KUKA KRL program: MyProgram_308().src

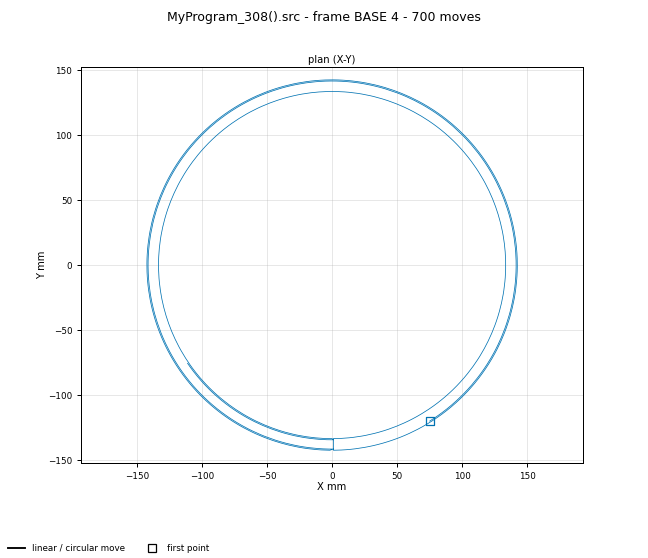
[picture p0: tool path of MyProgram_308().src in frame BASE 4, 700 of 700 moves have a stored position in this frame; points joined in program order, loops and branches not executed]
&ACCESS RVP
&REL 1
&PARAM TEMPLATE = C:\KRC\Roboter\Template\vorgabe
&PARAM EDITMASK = *
DEF MyProgram_308()
; ---- Setting reference (Base) ----
$BASE = BASE_DATA[4]

; --------------------------
; ---- Setting tool (TCP) ----
$TOOL = TOOL_DATA[3]
; --------------------------

$VEL.CP = VEL_APROX_PRINT
Startdeposition()
$VEL.CP = VEL_PRINT
LIN {X 75.0698,Y -120.0546,Z 181,A -53.2444,B 4.6912,C 0.3512,E1 4.792,E2 505.9034} C_DIS
LIN {X 78.7093,Y -117.7003,Z 181,A -51.6631,B 4.6912,C 0.3506,E1 4.7956,E2 504.3443} C_DIS
LIN {X 81.6771,Y -115.6604,Z 181,A -50.1341,B 4.6915,C 0.3471,E1 4.7991,E2 502.8043} C_DIS
LIN {X 84.8827,Y -113.3295,Z 181,A -48.4927,B 4.6918,C 0.3438,E1 4.8028,E2 501.1565} C_DIS
LIN {X 88.5091,Y -110.5206,Z 181,A -46.7634,B 4.6918,C 0.342,E1 4.8066,E2 499.443} C_DIS
LIN {X 91.7786,Y -107.8201,Z 181,A -44.9889,B 4.6922,C 0.338,E1 4.8104,E2 497.659} C_DIS
LIN {X 95.3898,Y -104.6393,Z 181,A -43.0975,B 4.6924,C 0.3349,E1 4.8143,E2 495.7737} C_DIS
LIN {X 98.6334,Y -101.5873,Z 181,A -41.3388,B 4.6926,C 0.3318,E1 4.8179,E2 494.0193} C_DIS
LIN {X 101.7844,Y -98.4298,Z 181,A -39.801,B 4.6926,C 0.3316,E1 4.8208,E2 492.5162} C_DIS
LIN {X 104.4298,Y -95.6189,Z 181,A -38.0744,B 4.693,C 0.326,E1 4.8242,E2 490.766} C_DIS
LIN {X 107.3448,Y -92.334,Z 181,A -36.3549,B 4.6932,C 0.3229,E1 4.8273,E2 489.0528} C_DIS
LIN {X 110.0788,Y -89.0572,Z 181,A -34.8071,B 4.6933,C 0.3214,E1 4.83,E2 487.5278} C_DIS
LIN {X 111.9572,Y -86.6838,Z 181,A -33.148,B 4.6939,C 0.3127,E1 4.833,E2 485.8087} C_DIS
LIN {X 114.3083,Y -83.5596,Z 181,A -31.9004,B 4.6939,C 0.3136,E1 4.8349,E2 484.6052} C_DIS
LIN {X 116.9623,Y -79.8026,Z 181,A -30.0572,B 4.6942,C 0.3094,E1 4.8379,E2 482.7628} C_DIS
LIN {X 119.4438,Y -76.0381,Z 181,A -28.3668,B 4.6943,C 0.3068,E1 4.8404,E2 481.0891} C_DIS
LIN {X 122.1556,Y -71.5997,Z 181,A -26.2713,B 4.6946,C 0.3017,E1 4.8434,E2 478.993} C_DIS
LIN {X 124.3843,Y -67.654,Z 181,A -24.4934,B 4.6949,C 0.2979,E1 4.8458,E2 477.2211} C_DIS
LIN {X 125.8992,Y -64.7895,Z 181,A -23.2049,B 4.6951,C 0.2948,E1 4.8475,E2 475.9344} C_DIS
LIN {X 127.5298,Y -61.5171,Z 181,A -21.7796,B 4.6953,C 0.2917,E1 4.8492,E2 474.5151} C_DIS
LIN {X 129.1189,Y -58.1061,Z 181,A -20.448,B 4.6953,C 0.2904,E1 4.8508,E2 473.2081} C_DIS
LIN {X 130.2583,Y -55.509,Z 181,A -19.102,B 4.6957,C 0.2846,E1 4.8523,E2 471.8344} C_DIS
LIN {X 131.8713,Y -51.5555,Z 181,A -17.5331,B 4.6959,C 0.2823,E1 4.8539,E2 470.2854} C_DIS
LIN {X 132.9031,Y -48.8412,Z 181,A -16.3204,B 4.6961,C 0.2786,E1 4.8551,E2 469.0666} C_DIS
LIN {X 134.269,Y -44.9427,Z 181,A -14.7391,B 4.6963,C 0.2753,E1 4.8565,E2 467.496} C_DIS
LIN {X 136.3041,Y -38.3301,Z 181,A -12.0529,B 4.6966,C 0.2692,E1 4.8586,E2 464.8228} C_DIS
LIN {X 137.081,Y -35.4568,Z 181,A -10.8532,B 4.6968,C 0.266,E1 4.8595,E2 463.6229} C_DIS
LIN {X 138.0053,Y -31.6629,Z 181,A -9.3753,B 4.697,C 0.263,E1 4.8604,E2 462.1573} C_DIS
LIN {X 138.7732,Y -28.1073,Z 181,A -7.5819,B 4.6974,C 0.2544,E1 4.8615,E2 460.3195} C_DIS
LIN {X 139.4952,Y -24.2805,Z 181,A -6.4089,B 4.6974,C 0.2557,E1 4.862,E2 459.1994} C_DIS
LIN {X 140.1291,Y -20.2963,Z 181,A -4.8304,B 4.6976,C 0.2518,E1 4.8627,E2 457.6269} C_DIS
LIN {X 140.5376,Y -17.2466,Z 181,A -3.7029,B 4.6976,C 0.2499,E1 4.8631,E2 456.514} C_DIS
LIN {X 140.9283,Y -13.6855,Z 181,A -2.1446,B 4.698,C 0.2443,E1 4.8635,E2 454.9401} C_DIS
LIN {X 141.2861,Y -9.3092,Z 181,A -0.4295,B 4.6982,C 0.2401,E1 4.8639,E2 453.232} C_DIS
LIN {X 141.4814,Y -5.5757,Z 181,A 1.0114,B 4.6984,C 0.2369,E1 4.864,E2 451.7995} C_DIS
LIN {X 141.586,Y -1.378,Z 181,A 2.7807,B 4.6986,C 0.231,E1 4.8641,E2 450.0196} C_DIS
LIN {X 141.5531,Y 3.3379,Z 181,A 4.462,B 4.6988,C 0.2288,E1 4.8641,E2 448.3671} C_DIS
LIN {X 141.4301,Y 6.7613,Z 181,A 5.8594,B 4.699,C 0.2247,E1 4.8639,E2 446.9673} C_DIS
LIN {X 141.2496,Y 9.8399,Z 181,A 6.9078,B 4.699,C 0.224,E1 4.8637,E2 445.9445} C_DIS
LIN {X 140.9695,Y 13.2561,Z 181,A 8.4681,B 4.6993,C 0.2176,E1 4.8633,E2 444.3602} C_DIS
LIN {X 140.3837,Y 18.4514,Z 181,A 10.3733,B 4.6994,C 0.2146,E1 4.8627,E2 442.4815} C_DIS
LIN {X 140.0089,Y 21.1151,Z 181,A 11.6157,B 4.6997,C 0.2094,E1 4.8622,E2 441.2181} C_DIS
LIN {X 139.3741,Y 24.9573,Z 181,A 12.9342,B 4.6997,C 0.2086,E1 4.8616,E2 439.9326} C_DIS
LIN {X 138.9009,Y 27.4798,Z 181,A 14.2341,B 4.7,C 0.2021,E1 4.8609,E2 438.5975} C_DIS
LIN {X 137.7792,Y 32.6373,Z 181,A 16.1101,B 4.7,C 0.1998,E1 4.8597,E2 436.7545} C_DIS
LIN {X 136.9433,Y 35.983,Z 181,A 17.4908,B 4.7002,C 0.1961,E1 4.8588,E2 435.375} C_DIS
LIN {X 135.9497,Y 39.5689,Z 181,A 18.9903,B 4.7004,C 0.1921,E1 4.8576,E2 433.8754} C_DIS
LIN {X 134.7946,Y 43.341,Z 181,A 20.5617,B 4.7006,C 0.1881,E1 4.8563,E2 432.3064} C_DIS
LIN {X 133.383,Y 47.5102,Z 181,A 22.24,B 4.7006,C 0.1848,E1 4.8548,E2 430.6407} C_DIS
LIN {X 132.4041,Y 50.1735,Z 181,A 23.4858,B 4.7009,C 0.1804,E1 4.8535,E2 429.3815} C_DIS
LIN {X 130.8136,Y 54.184,Z 181,A 25.0802,B 4.7009,C 0.1779,E1 4.8519,E2 427.8061} C_DIS
LIN {X 129.2904,Y 57.7228,Z 181,A 26.5611,B 4.7011,C 0.1749,E1 4.8502,E2 426.3346} C_DIS
LIN {X 127.7587,Y 61.038,Z 181,A 27.9434,B 4.7011,C 0.1724,E1 4.8486,E2 424.9642} C_DIS
LIN {X 126.5593,Y 63.4928,Z 181,A 29.1321,B 4.7013,C 0.1684,E1 4.8471,E2 423.7642} C_DIS
LIN {X 124.5791,Y 67.2951,Z 181,A 30.7949,B 4.7014,C 0.165,E1 4.8449,E2 422.1101} C_DIS
LIN {X 122.3445,Y 71.2774,Z 181,A 32.6523,B 4.7016,C 0.1604,E1 4.8424,E2 420.2507} C_DIS
LIN {X 119.9551,Y 75.2291,Z 181,A 34.4946,B 4.7017,C 0.1562,E1 4.8397,E2 418.4111} C_DIS
LIN {X 117.6471,Y 78.7889,Z 181,A 36.1286,B 4.7018,C 0.1532,E1 4.8372,E2 416.7873} C_DIS
LIN {X 114.9795,Y 82.6336,Z 181,A 37.9619,B 4.7019,C 0.1496,E1 4.8342,E2 414.9613} C_DIS
LIN {X 112.2893,Y 86.2536,Z 181,A 39.6305,B 4.702,C 0.1475,E1 4.8315,E2 413.3125} C_DIS
LIN {X 106.5861,Y 93.2089,Z 181,A 43.4318,B 4.7023,C 0.1374,E1 4.8246,E2 409.4894} C_DIS
LIN {X 103.0849,Y 97.067,Z 181,A 45.3479,B 4.7023,C 0.1355,E1 4.821,E2 407.5978} C_DIS
LIN {X 100.0737,Y 100.1693,Z 181,A 46.8348,B 4.7023,C 0.1353,E1 4.8182,E2 406.1446} C_DIS
LIN {X 93.3224,Y 106.4871,Z 181,A 50.5417,B 4.7026,C 0.1285,E1 4.8106,E2 402.4419} C_DIS
LIN {X 90.1706,Y 109.1685,Z 181,A 52.3912,B 4.7027,C 0.1231,E1 4.8066,E2 400.5697} C_DIS
LIN {X 86.5348,Y 112.0727,Z 181,A 54.2486,B 4.7027,C 0.1201,E1 4.8025,E2 398.7154} C_DIS
LIN {X 83.8855,Y 114.0689,Z 181,A 55.5799,B 4.7028,C 0.1179,E1 4.7996,E2 397.3854} C_DIS
LIN {X 80.2008,Y 116.689,Z 181,A 57.3008,B 4.7028,C 0.1162,E1 4.7956,E2 395.6784} C_DIS
LIN {X 76.9077,Y 118.8854,Z 181,A 58.9355,B 4.703,C 0.1132,E1 4.7918,E2 394.0395} C_DIS
LIN {X 72.9949,Y 121.3274,Z 181,A 60.7925,B 4.703,C 0.1105,E1 4.7874,E2 392.1836} C_DIS
LIN {X 69.2396,Y 123.5087,Z 181,A 62.451,B 4.703,C 0.1092,E1 4.7834,E2 390.5379} C_DIS
LIN {X 63.3482,Y 126.6315,Z 181,A 65.2652,B 4.7032,C 0.1042,E1 4.7764,E2 387.709} C_DIS
LIN {X 59.7789,Y 128.3532,Z 181,A 66.6825,B 4.7032,C 0.1044,E1 4.7729,E2 386.3158} C_DIS
LIN {X 56.9567,Y 129.6324,Z 181,A 68.0491,B 4.7032,C 0.1015,E1 4.7693,E2 384.9349} C_DIS
LIN {X 53.1414,Y 131.2401,Z 181,A 69.5466,B 4.7032,C 0.1017,E1 4.7655,E2 383.4604} C_DIS
LIN {X 49.8744,Y 132.5162,Z 181,A 70.9201,B 4.7032,C 0.1008,E1 4.762,E2 382.093} C_DIS
LIN {X 40.9953,Y 135.5269,Z 181,A 74.8213,B 4.7033,C 0.096,E1 4.7516,E2 378.179} C_DIS
LIN {X 36.8931,Y 136.7006,Z 181,A 76.5078,B 4.7033,C 0.095,E1 4.7471,E2 376.4981} C_DIS
LIN {X 33.4054,Y 137.594,Z 181,A 77.7795,B 4.7033,C 0.096,E1 4.7437,E2 375.2504} C_DIS
LIN {X 30.6843,Y 138.2285,Z 181,A 79.1401,B 4.7034,C 0.0927,E1 4.7399,E2 373.8608} C_DIS
LIN {X 26.746,Y 139.042,Z 181,A 80.4923,B 4.7034,C 0.0948,E1 4.7363,E2 372.5442} C_DIS
LIN {X 23.8286,Y 139.5725,Z 181,A 81.677,B 4.7034,C 0.0943,E1 4.733,E2 371.3618} C_DIS
LIN {X 19.8304,Y 140.1956,Z 181,A 83.4833,B 4.7034,C 0.0916,E1 4.728,E2 369.5344} C_DIS
LIN {X 15.3119,Y 140.7608,Z 181,A 85.3214,B 4.7034,C 0.091,E1 4.7229,E2 367.6976} C_DIS
LIN {X 11.0147,Y 141.1638,Z 181,A 87.1046,B 4.7034,C 0.09,E1 4.7179,E2 365.9104} C_DIS
LIN {X 7.1187,Y 141.4121,Z 181,A 88.5972,B 4.7034,C 0.0906,E1 4.7138,E2 364.4296} C_DIS
LIN {X 3.2569,Y 141.5554,Z 181,A 90.2585,B 4.7034,C 0.0894,E1 4.7091,E2 362.7565} C_DIS
LIN {X -0.7627,Y 141.5892,Z 181,A 91.8211,B 4.7034,C 0.09,E1 4.7048,E2 361.2027} C_DIS
LIN {X -5.1735,Y 141.4971,Z 181,A 93.539,B 4.7034,C 0.0907,E1 4.7,E2 359.4942} C_DIS
LIN {X -9.289,Y 141.2873,Z 181,A 95.2117,B 4.7034,C 0.0908,E1 4.6953,E2 357.8217} C_DIS
LIN {X -12.5503,Y 141.0352,Z 181,A 96.6728,B 4.7034,C 0.0896,E1 4.6912,E2 356.3437} C_DIS
LIN {X -16.7152,Y 140.601,Z 181,A 98.1672,B 4.7034,C 0.0921,E1 4.6871,E2 354.8757} C_DIS
LIN {X -19.9485,Y 140.1788,Z 181,A 99.6568,B 4.7034,C 0.0908,E1 4.6829,E2 353.3651} C_DIS
LIN {X -26.656,Y 139.0592,Z 181,A 102.3603,B 4.7034,C 0.0925,E1 4.6755,E2 350.6693} C_DIS
LIN {X -30.8555,Y 138.1897,Z 181,A 104.1566,B 4.7034,C 0.0928,E1 4.6706,E2 348.8663} C_DIS
LIN {X -34.9302,Y 137.2147,Z 181,A 106.2055,B 4.7034,C 0.0904,E1 4.6649,E2 346.7731} C_DIS
LIN {X -38.9949,Y 136.1177,Z 181,A 107.6813,B 4.7034,C 0.0939,E1 4.661,E2 345.3277} C_DIS
LIN {X -42.9866,Y 134.9078,Z 181,A 109.1542,B 4.7034,C 0.0973,E1 4.6572,E2 343.8832} C_DIS
LIN {X -45.9624,Y 133.9239,Z 181,A 110.5613,B 4.7034,C 0.0971,E1 4.6534,E2 342.4592} C_DIS
LIN {X -50.6433,Y 132.2259,Z 181,A 112.6753,B 4.7033,C 0.098,E1 4.6479,E2 340.3338} C_DIS
LIN {X -55.2956,Y 130.3492,Z 181,A 114.6914,B 4.7033,C 0.1003,E1 4.6427,E2 338.321} C_DIS
LIN {X -58.987,Y 128.7194,Z 181,A 116.2274,B 4.7032,C 0.103,E1 4.6388,E2 336.7984} C_DIS
LIN {X -62.3316,Y 127.133,Z 181,A 117.8537,B 4.7032,C 0.1036,E1 4.6347,E2 335.1568} C_DIS
LIN {X -65.869,Y 125.3362,Z 181,A 119.3462,B 4.7032,C 0.1066,E1 4.631,E2 333.6798} C_DIS
LIN {X -69.7137,Y 123.2422,Z 181,A 121.3293,B 4.7031,C 0.1071,E1 4.6261,E2 331.671} C_DIS
LIN {X -73.2602,Y 121.167,Z 181,A 123.0811,B 4.7031,C 0.1086,E1 4.6219,E2 329.9091} C_DIS
LIN {X -77.419,Y 118.5535,Z 181,A 124.9858,B 4.703,C 0.1124,E1 4.6174,E2 328.0165} C_DIS
LIN {X -81.0355,Y 116.111,Z 181,A 127.4359,B 4.703,C 0.1091,E1 4.6116,E2 325.4796} C_DIS
LIN {X -85.8049,Y 112.6324,Z 181,A 129.1986,B 4.7028,C 0.1186,E1 4.6079,E2 323.7996} C_DIS
LIN {X -89.309,Y 109.875,Z 181,A 131.0778,B 4.7028,C 0.1211,E1 4.6037,E2 321.9122} C_DIS
LIN {X -94.0851,Y 105.8142,Z 181,A 133.7725,B 4.7027,C 0.1244,E1 4.598,E2 319.1993} C_DIS
LIN {X -97.8206,Y 102.3699,Z 181,A 135.7338,B 4.7025,C 0.1291,E1 4.594,E2 317.2518} C_DIS
LIN {X -101.0745,Y 99.1586,Z 181,A 137.4276,B 4.7025,C 0.1341,E1 4.5907,E2 315.5796} C_DIS
LIN {X -104.3645,Y 95.6897,Z 181,A 139.7639,B 4.7024,C 0.1348,E1 4.5862,E2 313.1933} C_DIS
LIN {X -108.9183,Y 90.4728,Z 181,A 142.4907,B 4.7022,C 0.1414,E1 4.5813,E2 310.4785} C_DIS
LIN {X -111.3815,Y 87.4222,Z 181,A 144.7144,B 4.7022,C 0.1397,E1 4.5773,E2 308.1735} C_DIS
LIN {X -114.7727,Y 82.9202,Z 181,A 146.4482,B 4.7019,C 0.1493,E1 4.5746,E2 306.5127} C_DIS
LIN {X -117.5085,Y 78.9965,Z 181,A 148.4309,B 4.7019,C 0.1535,E1 4.5714,E2 304.5256} C_DIS
LIN {X -119.9878,Y 75.1771,Z 181,A 150.3081,B 4.7017,C 0.1576,E1 4.5686,E2 302.6455} C_DIS
LIN {X -122.2793,Y 71.3892,Z 181,A 152.1606,B 4.7015,C 0.1615,E1 4.566,E2 300.7867} C_DIS
LIN {X -124.544,Y 67.3605,Z 181,A 154.2725,B 4.7015,C 0.1642,E1 4.5631,E2 298.645} C_DIS
LIN {X -127.5781,Y 61.416,Z 181,A 156.8039,B 4.7012,C 0.1724,E1 4.56,E2 296.1378} C_DIS
LIN {X -129.1557,Y 58.0239,Z 181,A 158.2666,B 4.701,C 0.1767,E1 4.5583,E2 294.6829} C_DIS
LIN {X -130.6168,Y 54.6552,Z 181,A 160.1469,B 4.701,C 0.1775,E1 4.5562,E2 292.7526} C_DIS
LIN {X -131.8967,Y 51.49,Z 181,A 161.1438,B 4.7007,C 0.1841,E1 4.5552,E2 291.8069} C_DIS
LIN {X -133.1869,Y 48.0541,Z 181,A 162.6936,B 4.7006,C 0.1876,E1 4.5537,E2 290.25} C_DIS
LIN {X -134.2123,Y 45.1128,Z 181,A 164.1152,B 4.7005,C 0.1897,E1 4.5524,E2 288.8085} C_DIS
LIN {X -135.1278,Y 42.298,Z 181,A 165.46,B 4.7005,C 0.1919,E1 4.5512,E2 287.4456} C_DIS
LIN {X -136.2771,Y 38.4268,Z 181,A 166.9406,B 4.7002,C 0.1975,E1 4.5501,E2 285.9863} C_DIS
LIN {X -137.0595,Y 35.5416,Z 181,A 168.2933,B 4.7001,C 0.1997,E1 4.5491,E2 284.616} C_DIS
LIN {X -137.9376,Y 31.9593,Z 181,A 169.7965,B 4.6999,C 0.2038,E1 4.5482,E2 283.1126} C_DIS
LIN {X -139.6077,Y 23.6179,Z 181,A 173.2482,B 4.6995,C 0.2133,E1 4.5463,E2 279.6626} C_DIS
LIN {X -140.1454,Y 20.1817,Z 181,A 174.8493,B 4.6994,C 0.2158,E1 4.5456,E2 278.0372} C_DIS
LIN {X -140.5978,Y 16.7416,Z 181,A 176.4714,B 4.6993,C 0.2181,E1 4.5451,E2 276.3877} C_DIS
LIN {X -141.1395,Y 11.3155,Z 181,A 178.4973,B 4.6989,C 0.2257,E1 4.5446,E2 274.3872} C_DIS
LIN {X -141.3929,Y 7.5008,Z 181,A -179.7628,B 4.6988,C 0.2286,E1 4.5443,E2 272.6231} C_DIS
LIN {X -141.5554,Y 3.2567,Z 181,A -178.0314,B 4.6985,C 0.2334,E1 4.5441,E2 270.8914} C_DIS
LIN {X -141.5872,Y -1.1633,Z 181,A -176.0293,B 4.6984,C 0.2368,E1 4.5441,E2 268.8624} C_DIS
LIN {X -141.4468,Y -6.4295,Z 181,A -173.9597,B 4.698,C 0.2434,E1 4.5444,E2 266.8026} C_DIS
LIN {X -141.2321,Y -10.0803,Z 181,A -172.5422,B 4.6978,C 0.248,E1 4.5446,E2 265.3943} C_DIS
LIN {X -140.7433,Y -15.4747,Z 181,A -170.1247,B 4.6975,C 0.2525,E1 4.5453,E2 262.9485} C_DIS
LIN {X -139.8187,Y -22.3429,Z 181,A -167.2867,B 4.6971,C 0.2601,E1 4.5464,E2 260.108} C_DIS
LIN {X -138.8155,Y -27.8994,Z 181,A -165.0707,B 4.6967,C 0.267,E1 4.5476,E2 257.9025} C_DIS
LIN {X -138.0973,Y -31.2601,Z 181,A -163.5807,B 4.6966,C 0.27,E1 4.5485,E2 256.4002} C_DIS
LIN {X -137.3318,Y -34.4688,Z 181,A -162.248,B 4.6964,C 0.2737,E1 4.5493,E2 255.0686} C_DIS
LIN {X -136.4961,Y -37.6438,Z 181,A -160.7575,B 4.6962,C 0.276,E1 4.5504,E2 253.5574} C_DIS
LIN {X -135.3678,Y -41.5155,Z 181,A -159.2211,B 4.6959,C 0.2812,E1 4.5517,E2 252.0346} C_DIS
LIN {X -134.4688,Y -44.3426,Z 181,A -157.895,B 4.6958,C 0.2834,E1 4.5528,E2 250.6925} C_DIS
LIN {X -131.6285,Y -52.1779,Z 181,A -154.3869,B 4.6953,C 0.2912,E1 4.5563,E2 247.1683} C_DIS
LIN {X -130.1111,Y -55.8495,Z 181,A -152.8289,B 4.695,C 0.2958,E1 4.5579,E2 245.6176} C_DIS
LIN {X -128.1677,Y -60.18,Z 181,A -150.6827,B 4.6948,C 0.2989,E1 4.5605,E2 243.4424} C_DIS
LIN {X -126.466,Y -63.6761,Z 181,A -149.1337,B 4.6946,C 0.303,E1 4.5624,E2 241.8972} C_DIS
LIN {X -124.9855,Y -66.5369,Z 181,A -147.4561,B 4.6946,C 0.3031,E1 4.5647,E2 240.1701} C_DIS
LIN {X -123.0449,Y -70.0604,Z 181,A -146.1359,B 4.6941,C 0.3096,E1 4.5664,E2 238.8919} C_DIS
LIN {X -120.894,Y -73.7108,Z 181,A -144.3196,B 4.6939,C 0.3129,E1 4.569,E2 237.0626} C_DIS
LIN {X -118.2629,Y -77.8612,Z 181,A -142.3417,B 4.6936,C 0.3176,E1 4.572,E2 235.0869} C_DIS
LIN {X -115.7411,Y -81.5627,Z 181,A -140.4547,B 4.6934,C 0.3211,E1 4.575,E2 233.1905} C_DIS
LIN {X -113.044,Y -85.2616,Z 181,A -138.5665,B 4.6931,C 0.3249,E1 4.5782,E2 231.2981} C_DIS
LIN {X -110.2585,Y -88.8344,Z 181,A -136.6725,B 4.6929,C 0.3283,E1 4.5815,E2 229.3964} C_DIS
LIN {X -107.2744,Y -92.4158,Z 181,A -134.7539,B 4.6926,C 0.332,E1 4.585,E2 227.474} C_DIS
LIN {X -104.2592,Y -95.8045,Z 181,A -132.8957,B 4.6924,C 0.3356,E1 4.5885,E2 225.6132} C_DIS
LIN {X -101.5601,Y -98.6615,Z 181,A -131.1972,B 4.6922,C 0.3377,E1 4.5918,E2 223.9004} C_DIS
LIN {X -98.3525,Y -101.8592,Z 181,A -129.3937,B 4.6919,C 0.3415,E1 4.5954,E2 222.1011} C_DIS
LIN {X -95.0209,Y -104.974,Z 181,A -127.5142,B 4.6917,C 0.3446,E1 4.5992,E2 220.2173} C_DIS
LIN {X -91.5976,Y -107.974,Z 181,A -125.6499,B 4.6915,C 0.3477,E1 4.6032,E2 218.3503} C_DIS
LIN {X -88.1064,Y -110.8411,Z 181,A -123.7504,B 4.6913,C 0.3501,E1 4.6073,E2 216.4413} C_DIS
LIN {X -84.0911,Y -113.9178,Z 181,A -121.6429,B 4.6911,C 0.3528,E1 4.6121,E2 214.3257} C_DIS
LIN {X -80.5702,Y -116.4348,Z 181,A -119.8851,B 4.6909,C 0.3555,E1 4.6161,E2 212.5672} C_DIS
LIN {X -76.9874,Y -118.8337,Z 181,A -118.177,B 4.6907,C 0.3584,E1 4.62,E2 210.8641} C_DIS
LIN {X -73.5376,Y -120.9992,Z 181,A -116.4192,B 4.6906,C 0.3596,E1 4.6243,E2 209.0914} C_DIS
LIN {X -69.5855,Y -123.3143,Z 181,A -114.3926,B 4.6906,C 0.3603,E1 4.6292,E2 207.041} C_DIS
LIN {X -64.7433,Y -125.9227,Z 181,A -112.4191,B 4.6901,C 0.3655,E1 4.634,E2 205.1018} C_DIS
LIN {X -61.4276,Y -127.5725,Z 181,A -110.867,B 4.6901,C 0.3667,E1 4.6379,E2 203.5422} C_DIS
LIN {X -58.1448,Y -129.1017,Z 181,A -109.4689,B 4.6899,C 0.3689,E1 4.6415,E2 202.1531} C_DIS
LIN {X -54.9998,Y -130.4729,Z 181,A -108.0234,B 4.6898,C 0.3697,E1 4.6452,E2 200.6997} C_DIS
LIN {X -51.6876,Y -131.82,Z 181,A -106.6986,B 4.6896,C 0.3723,E1 4.6486,E2 199.3913} C_DIS
LIN {X -43.683,Y -134.685,Z 181,A -102.9647,B 4.6896,C 0.3722,E1 4.6586,E2 195.6169} C_DIS
LIN {X -40.093,Y -135.7962,Z 181,A -101.4824,B 4.6895,C 0.3736,E1 4.6625,E2 194.1396} C_DIS
LIN {X -35.6163,Y -137.0405,Z 181,A -99.66,B 4.6893,C 0.3754,E1 4.6674,E2 192.3247} C_DIS
LIN {X -31.8927,Y -137.9528,Z 181,A -98.073,B 4.6893,C 0.3758,E1 4.6717,E2 190.7322} C_DIS
LIN {X -28.8624,Y -138.6195,Z 181,A -96.8968,B 4.6892,C 0.3772,E1 4.6749,E2 189.5665} C_DIS
LIN {X -25.2409,Y -139.3234,Z 181,A -95.273,B 4.6892,C 0.3764,E1 4.6794,E2 187.9243} C_DIS
LIN {X -21.4469,Y -139.9575,Z 181,A -93.7514,B 4.6892,C 0.3773,E1 4.6836,E2 186.407} C_DIS
LIN {X -17.2173,Y -140.5411,Z 181,A -91.9833,B 4.6892,C 0.3773,E1 4.6885,E2 184.6328} C_DIS
LIN {X -13.7723,Y -140.9199,Z 181,A -90.6643,B 4.6892,C 0.3784,E1 4.6921,E2 183.3246} C_DIS
LIN {X -10.6013,Y -141.194,Z 181,A -89.3284,B 4.6892,C 0.378,E1 4.6959,E2 181.9817} C_DIS
LIN {X -6.9612,Y -141.42,Z 181,A -87.8113,B 4.6892,C 0.3776,E1 4.7001,E2 180.4583} C_DIS
LIN {X -2.4965,Y -141.5693,Z 181,A -86.169,B 4.689,C 0.3793,E1 4.7047,E2 178.8378} C_DIS
LIN {X 1.0182,Y -141.5859,Z 181,A -84.7274,B 4.689,C 0.3789,E1 4.7087,E2 177.3927} C_DIS
Enddeposition()
LIN {X 1.0182,Y -141.5859,Z 181,A -84.7274,B 4.689,C 0.3789,E1 4.7087,E2 177.3927} C_DIS
Startdeposition()
$VEL.CP = VEL_PRINT
LIN {X -1.746,Y -142.4843,Z 181,A -86.2389,B 4.6888,C 0.3862,E1 4.7045,E2 178.9914} C_DIS
LIN {X -4.7667,Y -142.416,Z 181,A -87.672,B 4.6885,C 0.3887,E1 4.7004,E2 180.4548} C_DIS
LIN {X -8.2577,Y -142.255,Z 181,A -89.0045,B 4.6886,C 0.3879,E1 4.6967,E2 181.778} C_DIS
LIN {X -12.2264,Y -141.9682,Z 181,A -90.5419,B 4.6886,C 0.387,E1 4.6925,E2 183.3075} C_DIS
LIN {X -15.7037,Y -141.6262,Z 181,A -91.9458,B 4.6887,C 0.3868,E1 4.6886,E2 184.7118} C_DIS
LIN {X -19.172,Y -141.1993,Z 181,A -93.3519,B 4.6887,C 0.3865,E1 4.6847,E2 186.1185} C_DIS
LIN {X -22.1602,Y -140.7601,Z 181,A -94.5771,B 4.6887,C 0.3862,E1 4.6813,E2 187.3456} C_DIS
LIN {X -26.0839,Y -140.0873,Z 181,A -96.1982,B 4.6887,C 0.3859,E1 4.6768,E2 188.97} C_DIS
LIN {X -29.5094,Y -139.4054,Z 181,A -97.6066,B 4.6888,C 0.3853,E1 4.673,E2 190.3794} C_DIS
LIN {X -32.9167,Y -138.64,Z 181,A -99.0165,B 4.6888,C 0.3846,E1 4.6691,E2 191.7905} C_DIS
LIN {X -36.3044,Y -137.7915,Z 181,A -100.4286,B 4.6889,C 0.3839,E1 4.6653,E2 193.204} C_DIS
LIN {X -39.2247,Y -136.9907,Z 181,A -101.6544,B 4.6889,C 0.3832,E1 4.662,E2 194.4313} C_DIS
LIN {X -42.5646,Y -135.9899,Z 181,A -103.1792,B 4.6889,C 0.3835,E1 4.6579,E2 195.9732} C_DIS
LIN {X -45.8685,Y -134.9115,Z 181,A -104.4732,B 4.6891,C 0.3814,E1 4.6545,E2 197.2535} C_DIS
LIN {X -49.5405,Y -133.6048,Z 181,A -105.9139,B 4.6894,C 0.3787,E1 4.6507,E2 198.6772} C_DIS
LIN {X -52.4675,Y -132.4847,Z 181,A -107.4597,B 4.6892,C 0.3805,E1 4.6466,E2 200.2621} C_DIS
LIN {X -55.7022,Y -131.1574,Z 181,A -108.7515,B 4.6894,C 0.378,E1 4.6433,E2 201.5386} C_DIS
LIN {X -58.5454,Y -129.911,Z 181,A -110.0149,B 4.6895,C 0.3768,E1 4.6401,E2 202.8041} C_DIS
LIN {X -61.7106,Y -128.4374,Z 181,A -111.4353,B 4.6896,C 0.3754,E1 4.6365,E2 204.2269} C_DIS
LIN {X -64.8385,Y -126.8868,Z 181,A -112.8049,B 4.6898,C 0.3735,E1 4.6331,E2 205.5921} C_DIS
LIN {X -67.9132,Y -125.2708,Z 181,A -114.3873,B 4.6898,C 0.3735,E1 4.6291,E2 207.1997} C_DIS
LIN {X -71.5447,Y -123.2324,Z 181,A -116.0024,B 4.69,C 0.3708,E1 4.6252,E2 208.8069} C_DIS
LIN {X -75.2155,Y -121.0268,Z 181,A -117.8056,B 4.6901,C 0.3692,E1 4.6209,E2 210.6211} C_DIS
LIN {X -79.1656,Y -118.4806,Z 181,A -119.7432,B 4.6903,C 0.3669,E1 4.6164,E2 212.5651} C_DIS
LIN {X -82.7578,Y -116,Z 181,A -121.5247,B 4.6905,C 0.3645,E1 4.6123,E2 214.35} C_DIS
LIN {X -86.2739,Y -113.4098,Z 181,A -123.3317,B 4.6907,C 0.3621,E1 4.6082,E2 216.1638} C_DIS
LIN {X -89.9064,Y -110.5522,Z 181,A -125.2207,B 4.6909,C 0.3593,E1 4.6041,E2 218.0567} C_DIS
LIN {X -93.5528,Y -107.4837,Z 181,A -127.1646,B 4.6911,C 0.3561,E1 4.6,E2 220.0041} C_DIS
LIN {X -97.161,Y -104.2333,Z 181,A -129.1536,B 4.6914,C 0.3529,E1 4.5959,E2 221.9977} C_DIS
LIN {X -100.5656,Y -100.9526,Z 181,A -131.0742,B 4.6916,C 0.3494,E1 4.592,E2 223.9206} C_DIS
LIN {X -103.6383,Y -97.7954,Z 181,A -132.8382,B 4.6919,C 0.3459,E1 4.5886,E2 225.6832} C_DIS
LIN {X -106.5873,Y -94.5729,Z 181,A -134.6403,B 4.6921,C 0.3427,E1 4.5852,E2 227.491} C_DIS
LIN {X -109.0076,Y -91.7727,Z 181,A -136.234,B 4.6923,C 0.3405,E1 4.5823,E2 229.0985} C_DIS
LIN {X -111.7966,Y -88.3545,Z 181,A -138.0597,B 4.6925,C 0.3371,E1 4.5791,E2 230.9306} C_DIS
LIN {X -114.5935,Y -84.6955,Z 181,A -139.9151,B 4.6928,C 0.3331,E1 4.576,E2 232.7859} C_DIS
LIN {X -117.1386,Y -81.1386,Z 181,A -141.7535,B 4.6931,C 0.3297,E1 4.573,E2 234.6344} C_DIS
LIN {X -119.7917,Y -77.1683,Z 181,A -143.653,B 4.6934,C 0.3251,E1 4.5701,E2 236.5305} C_DIS
LIN {X -122.0978,Y -73.4647,Z 181,A -145.4926,B 4.6936,C 0.3217,E1 4.5674,E2 238.3807} C_DIS
LIN {X -124.4056,Y -69.4854,Z 181,A -147.3461,B 4.6939,C 0.3172,E1 4.5648,E2 240.234} C_DIS
LIN {X -126.4844,Y -65.6235,Z 181,A -149.1194,B 4.6942,C 0.3129,E1 4.5625,E2 242.0078} C_DIS
LIN {X -128.0554,Y -62.5014,Z 181,A -150.562,B 4.6944,C 0.3097,E1 4.5607,E2 243.4547} C_DIS
LIN {X -129.5539,Y -59.3322,Z 181,A -152.0579,B 4.6946,C 0.3068,E1 4.559,E2 244.9614} C_DIS
LIN {X -131.3317,Y -55.285,Z 181,A -153.983,B 4.6948,C 0.3034,E1 4.5568,E2 246.9052} C_DIS
LIN {X -132.9373,Y -51.3039,Z 181,A -155.611,B 4.6952,C 0.2982,E1 4.5552,E2 248.5193} C_DIS
LIN {X -134.1527,Y -48.0359,Z 181,A -157.0583,B 4.6954,C 0.2948,E1 4.5538,E2 249.9719} C_DIS
LIN {X -135.3018,Y -44.6971,Z 181,A -158.5156,B 4.6956,C 0.2913,E1 4.5525,E2 251.4333} C_DIS
LIN {X -136.357,Y -41.3666,Z 181,A -160.0023,B 4.6958,C 0.2882,E1 4.5512,E2 252.9301} C_DIS
LIN {X -137.664,Y -36.7826,Z 181,A -161.9393,B 4.6961,C 0.2831,E1 4.5498,E2 254.8687} C_DIS
LIN {X -138.5268,Y -33.3866,Z 181,A -163.3891,B 4.6963,C 0.2796,E1 4.5488,E2 256.3231} C_DIS
LIN {X -139.3041,Y -29.9787,Z 181,A -164.8369,B 4.6965,C 0.2761,E1 4.5479,E2 257.7755} C_DIS
LIN {X -140.001,Y -26.5353,Z 181,A -166.2894,B 4.6967,C 0.2724,E1 4.5471,E2 259.2325} C_DIS
LIN {X -140.6842,Y -22.6488,Z 181,A -167.933,B 4.6969,C 0.2685,E1 4.5464,E2 260.8826} C_DIS
LIN {X -141.1296,Y -19.6737,Z 181,A -169.1676,B 4.6971,C 0.2653,E1 4.5459,E2 262.1197} C_DIS
LIN {X -141.5704,Y -16.2067,Z 181,A -170.6116,B 4.6973,C 0.2616,E1 4.5454,E2 263.5678} C_DIS
LIN {X -141.9259,Y -12.7267,Z 181,A -172.1042,B 4.6975,C 0.2583,E1 4.545,E2 265.0708} C_DIS
LIN {X -142.1959,Y -9.2158,Z 181,A -173.6403,B 4.6977,C 0.2552,E1 4.5447,E2 266.6216} C_DIS
LIN {X -142.3968,Y -5.26,Z 181,A -175.1699,B 4.698,C 0.2502,E1 4.5445,E2 268.1418} C_DIS
LIN {X -142.4839,Y -1.7679,Z 181,A -176.6153,B 4.6981,C 0.2466,E1 4.5445,E2 269.5916} C_DIS
LIN {X -142.4907,Y 0.9319,Z 181,A -177.7816,B 4.6983,C 0.2441,E1 4.5445,E2 270.7677} C_DIS
LIN {X -142.4164,Y 4.7556,Z 181,A -179.4761,B 4.6984,C 0.2409,E1 4.5445,E2 272.4816} C_DIS
LIN {X -142.255,Y 8.2572,Z 181,A 179.1005,B 4.6986,C 0.237,E1 4.5448,E2 273.9057} C_DIS
LIN {X -141.9697,Y 12.2085,Z 181,A 177.5708,B 4.6989,C 0.232,E1 4.5451,E2 275.4259} C_DIS
LIN {X -141.6282,Y 15.6855,Z 181,A 176.1236,B 4.6991,C 0.2284,E1 4.5455,E2 276.8776} C_DIS
LIN {X -141.1993,Y 19.172,Z 181,A 174.6715,B 4.6992,C 0.2247,E1 4.546,E2 278.3338} C_DIS
LIN {X -140.761,Y 22.1545,Z 181,A 173.4143,B 4.6994,C 0.2216,E1 4.5466,E2 279.5959} C_DIS
LIN {X -140.094,Y 26.0488,Z 181,A 171.7583,B 4.6996,C 0.2177,E1 4.5474,E2 281.2595} C_DIS
LIN {X -139.4116,Y 29.4809,Z 181,A 170.4182,B 4.6998,C 0.2133,E1 4.5481,E2 282.5896} C_DIS
LIN {X -138.7287,Y 32.5481,Z 181,A 168.8993,B 4.6998,C 0.2117,E1 4.5491,E2 284.1408} C_DIS
LIN {X -137.6643,Y 36.7813,Z 181,A 167.1113,B 4.7,C 0.2071,E1 4.5503,E2 285.9315} C_DIS
LIN {X -136.4971,Y 40.9089,Z 181,A 165.4276,B 4.7003,C 0.2021,E1 4.5517,E2 287.6085} C_DIS
LIN {X -135.7023,Y 43.4649,Z 181,A 164.2167,B 4.7003,C 0.2002,E1 4.5527,E2 288.8359} C_DIS
LIN {X -134.5377,Y 46.9467,Z 181,A 162.8198,B 4.7005,C 0.1957,E1 4.5539,E2 290.2213} C_DIS
LIN {X -133.1183,Y 50.8381,Z 181,A 161.0884,B 4.7007,C 0.1917,E1 4.5556,E2 291.96} C_DIS
LIN {X -132.1247,Y 53.3606,Z 181,A 159.8706,B 4.7007,C 0.1899,E1 4.5569,E2 293.1932} C_DIS
LIN {X -130.4637,Y 57.3078,Z 181,A 158.1921,B 4.701,C 0.185,E1 4.5588,E2 294.8647} C_DIS
LIN {X -129.1909,Y 60.1174,Z 181,A 156.8444,B 4.701,C 0.1827,E1 4.5603,E2 296.2252} C_DIS
LIN {X -127.395,Y 63.84,Z 181,A 155.1987,B 4.7012,C 0.1783,E1 4.5624,E2 297.8676} C_DIS
LIN {X -125.793,Y 66.9401,Z 181,A 153.83,B 4.7014,C 0.1745,E1 4.5641,E2 299.2306} C_DIS
LIN {X -123.9841,Y 70.235,Z 181,A 152.0818,B 4.7014,C 0.1726,E1 4.5665,E2 301.008} C_DIS
LIN {X -121.7727,Y 74.0024,Z 181,A 150.2826,B 4.7016,C 0.1687,E1 4.5691,E2 302.8112} C_DIS
LIN {X -119.3165,Y 77.9009,Z 181,A 148.3762,B 4.7017,C 0.1647,E1 4.572,E2 304.7229} C_DIS
LIN {X -116.6391,Y 81.8552,Z 181,A 146.4775,B 4.7019,C 0.1601,E1 4.575,E2 306.6173} C_DIS
LIN {X -114.0638,Y 85.4074,Z 181,A 144.6836,B 4.702,C 0.1563,E1 4.578,E2 308.4135} C_DIS
LIN {X -111.3992,Y 88.8542,Z 181,A 142.8561,B 4.7021,C 0.153,E1 4.5811,E2 310.2492} C_DIS
LIN {X -108.4797,Y 92.3959,Z 181,A 141.0034,B 4.7022,C 0.1491,E1 4.5845,E2 312.1013} C_DIS
LIN {X -105.6035,Y 95.67,Z 181,A 139.2031,B 4.7023,C 0.1458,E1 4.5878,E2 313.9063} C_DIS
LIN {X -102.5955,Y 98.8893,Z 181,A 137.3277,B 4.7024,C 0.1431,E1 4.5914,E2 315.7935} C_DIS
LIN {X -99.35,Y 102.1495,Z 181,A 135.4649,B 4.7025,C 0.1395,E1 4.5951,E2 317.6565} C_DIS
LIN {X -96.3525,Y 104.9811,Z 181,A 133.7413,B 4.7026,C 0.1369,E1 4.5987,E2 319.387} C_DIS
LIN {X -93.0917,Y 107.8832,Z 181,A 132.0592,B 4.7027,C 0.1331,E1 4.6022,E2 321.0583} C_DIS
LIN {X -89.9098,Y 110.5494,Z 181,A 130.3243,B 4.7027,C 0.1306,E1 4.6059,E2 322.8004} C_DIS
LIN {X -86.485,Y 113.2484,Z 181,A 128.5004,B 4.7028,C 0.1282,E1 4.61,E2 324.6318} C_DIS
LIN {X -82.9763,Y 115.8438,Z 181,A 126.7017,B 4.7029,C 0.1258,E1 4.6141,E2 326.4348} C_DIS
LIN {X -79.1616,Y 118.4832,Z 181,A 124.786,B 4.7029,C 0.1233,E1 4.6185,E2 328.3555} C_DIS
LIN {X -75.2403,Y 121.0113,Z 181,A 122.8868,B 4.703,C 0.1207,E1 4.623,E2 330.2562} C_DIS
LIN {X -71.2045,Y 123.4293,Z 181,A 121.0273,B 4.7031,C 0.1178,E1 4.6274,E2 332.1103} C_DIS
LIN {X -67.7342,Y 125.3676,Z 181,A 119.3081,B 4.7031,C 0.1167,E1 4.6317,E2 333.8436} C_DIS
LIN {X -64.0592,Y 127.2836,Z 181,A 117.7438,B 4.7032,C 0.1137,E1 4.6355,E2 335.3937} C_DIS
LIN {X -61.4932,Y 128.5412,Z 181,A 116.5207,B 4.7032,C 0.113,E1 4.6386,E2 336.6254} C_DIS
LIN {X -57.7463,Y 130.2684,Z 181,A 114.9037,B 4.7032,C 0.1108,E1 4.6427,E2 338.2359} C_DIS
LIN {X -54.5377,Y 131.6437,Z 181,A 113.485,B 4.7033,C 0.1094,E1 4.6464,E2 339.6556} C_DIS
LIN {X -51.2961,Y 132.9403,Z 181,A 112.0668,B 4.7033,C 0.1082,E1 4.6501,E2 341.0746} C_DIS
LIN {X -48.0228,Y 134.1574,Z 181,A 110.6473,B 4.7033,C 0.107,E1 4.6538,E2 342.4951} C_DIS
LIN {X -44.6977,Y 135.3016,Z 181,A 109.2222,B 4.7034,C 0.1059,E1 4.6576,E2 343.9208} C_DIS
LIN {X -40.9093,Y 136.497,Z 181,A 107.4702,B 4.7034,C 0.1062,E1 4.6623,E2 345.6915} C_DIS
LIN {X -36.7642,Y 137.6689,Z 181,A 105.8664,B 4.7034,C 0.1037,E1 4.6666,E2 347.2779} C_DIS
LIN {X -33.3855,Y 138.527,Z 181,A 104.4555,B 4.7034,C 0.1029,E1 4.6704,E2 348.6891} C_DIS
LIN {X -29.987,Y 139.3023,Z 181,A 103.046,B 4.7034,C 0.1022,E1 4.6742,E2 350.0987} C_DIS
LIN {X -26.5684,Y 139.9947,Z 181,A 101.6376,B 4.7034,C 0.1016,E1 4.6781,E2 351.5072} C_DIS
LIN {X -22.6623,Y 140.682,Z 181,A 100.0311,B 4.7035,C 0.1011,E1 4.6825,E2 353.1143} C_DIS
LIN {X -19.6485,Y 141.1332,Z 181,A 98.8127,B 4.7035,C 0.1006,E1 4.6859,E2 354.3312} C_DIS
LIN {X -16.1813,Y 141.5734,Z 181,A 97.4081,B 4.7035,C 0.1002,E1 4.6898,E2 355.735} C_DIS
LIN {X -12.704,Y 141.9278,Z 181,A 95.9693,B 4.7035,C 0.1002,E1 4.6938,E2 357.1773} C_DIS
LIN {X -9.221,Y 142.1956,Z 181,A 94.4781,B 4.7035,C 0.1009,E1 4.698,E2 358.6788} C_DIS
LIN {X -5.2445,Y 142.3974,Z 181,A 92.987,B 4.7035,C 0.0996,E1 4.7021,E2 360.1552} C_DIS
LIN {X -1.7514,Y 142.4842,Z 181,A 91.615,B 4.7035,C 0.0993,E1 4.7059,E2 361.5224} C_DIS
LIN {X 1.0001,Y 142.4903,Z 181,A 90.4484,B 4.7035,C 0.1,E1 4.7092,E2 362.6961} C_DIS
LIN {X 4.7654,Y 142.416,Z 181,A 88.8211,B 4.7035,C 0.1014,E1 4.7138,E2 364.3372} C_DIS
LIN {X 8.2637,Y 142.2546,Z 181,A 87.4427,B 4.7035,C 0.1014,E1 4.7176,E2 365.7113} C_DIS
LIN {X 12.223,Y 141.9685,Z 181,A 85.9619,B 4.7035,C 0.1006,E1 4.7217,E2 367.1768} C_DIS
LIN {X 15.6999,Y 141.6267,Z 181,A 84.5659,B 4.7035,C 0.101,E1 4.7256,E2 368.5712} C_DIS
LIN {X 19.1687,Y 141.1997,Z 181,A 83.1695,B 4.7035,C 0.1015,E1 4.7295,E2 369.966} C_DIS
LIN {X 22.1461,Y 140.7623,Z 181,A 81.9568,B 4.7035,C 0.1021,E1 4.7328,E2 371.1786} C_DIS
LIN {X 26.0798,Y 140.0881,Z 181,A 80.3499,B 4.7035,C 0.103,E1 4.7372,E2 372.7854} C_DIS
LIN {X 29.5045,Y 139.4065,Z 181,A 78.9578,B 4.7035,C 0.1038,E1 4.741,E2 374.1755} C_DIS
LIN {X 32.9115,Y 138.6413,Z 181,A 77.5662,B 4.7035,C 0.1046,E1 4.7448,E2 375.5652} C_DIS
LIN {X 36.7633,Y 137.6691,Z 181,A 75.8971,B 4.7034,C 0.1066,E1 4.7493,E2 377.2429} C_DIS
LIN {X 40.8487,Y 136.5152,Z 181,A 74.295,B 4.7034,C 0.1069,E1 4.7536,E2 378.8314} C_DIS
LIN {X 44.5345,Y 135.356,Z 181,A 72.8794,B 4.7034,C 0.1067,E1 4.7573,E2 380.229} C_DIS
LIN {X 47.5084,Y 134.3428,Z 181,A 71.5085,B 4.7034,C 0.1092,E1 4.761,E2 381.6135} C_DIS
LIN {X 50.8372,Y 133.1187,Z 181,A 70.0976,B 4.7033,C 0.1105,E1 4.7647,E2 383.0223} C_DIS
LIN {X 53.3478,Y 132.1299,Z 181,A 68.9316,B 4.7033,C 0.1127,E1 4.7677,E2 384.1983} C_DIS
LIN {X 57.3093,Y 130.463,Z 181,A 67.3166,B 4.7033,C 0.1133,E1 4.7718,E2 385.7988} C_DIS
LIN {X 60.128,Y 129.186,Z 181,A 66.0851,B 4.7032,C 0.1147,E1 4.775,E2 387.0285} C_DIS
LIN {X 63.2853,Y 127.6687,Z 181,A 64.6979,B 4.7032,C 0.1163,E1 4.7784,E2 388.4129} C_DIS
LIN {X 66.3716,Y 126.0916,Z 181,A 63.3343,B 4.7032,C 0.1178,E1 4.7818,E2 389.7724} C_DIS
LIN {X 70.2341,Y 123.9846,Z 181,A 61.4581,B 4.703,C 0.1216,E1 4.7864,E2 391.6624} C_DIS
LIN {X 74.0083,Y 121.7691,Z 181,A 59.7321,B 4.703,C 0.1238,E1 4.7905,E2 393.384} C_DIS
LIN {X 77.9044,Y 119.3142,Z 181,A 57.9087,B 4.703,C 0.1264,E1 4.7948,E2 395.2039} C_DIS
LIN {X 81.8502,Y 116.6426,Z 181,A 56.0983,B 4.7029,C 0.1282,E1 4.799,E2 397.0008} C_DIS
LIN {X 85.0345,Y 114.3415,Z 181,A 54.4863,B 4.7028,C 0.1313,E1 4.8026,E2 398.6171} C_DIS
LIN {X 88.8533,Y 111.3999,Z 181,A 52.6211,B 4.7027,C 0.1339,E1 4.8067,E2 400.4731} C_DIS
LIN {X 92.4135,Y 108.4648,Z 181,A 50.8226,B 4.7027,C 0.1366,E1 4.8105,E2 402.2645} C_DIS
LIN {X 95.0347,Y 106.1755,Z 181,A 49.4068,B 4.7025,C 0.1395,E1 4.8135,E2 403.6826} C_DIS
LIN {X 98.236,Y 103.2211,Z 181,A 47.6756,B 4.7025,C 0.1427,E1 4.817,E2 405.4116} C_DIS
LIN {X 101.3753,Y 100.1401,Z 181,A 46.0128,B 4.7024,C 0.1449,E1 4.8203,E2 407.061} C_DIS
LIN {X 104.3969,Y 96.9853,Z 181,A 44.2298,B 4.7022,C 0.1489,E1 4.8237,E2 408.8478} C_DIS
LIN {X 107.481,Y 93.5558,Z 181,A 42.419,B 4.7022,C 0.1523,E1 4.827,E2 410.6534} C_DIS
LIN {X 110.54,Y 89.9213,Z 181,A 40.629,B 4.702,C 0.1549,E1 4.8302,E2 412.4284} C_DIS
LIN {X 113.2377,Y 86.4988,Z 181,A 38.8733,B 4.702,C 0.1589,E1 4.8332,E2 414.1851} C_DIS
LIN {X 115.857,Y 82.9578,Z 181,A 37.1443,B 4.7018,C 0.1625,E1 4.8361,E2 415.9093} C_DIS
LIN {X 118.4819,Y 79.1636,Z 181,A 35.3144,B 4.7017,C 0.1665,E1 4.8389,E2 417.7365} C_DIS
LIN {X 120.8519,Y 75.4964,Z 181,A 33.5937,B 4.7015,C 0.1703,E1 4.8415,E2 419.4534} C_DIS
LIN {X 123.2283,Y 71.5517,Z 181,A 31.8099,B 4.7014,C 0.1739,E1 4.844,E2 421.229} C_DIS
LIN {X 125.3689,Y 67.7317,Z 181,A 30.0567,B 4.7012,C 0.1782,E1 4.8464,E2 422.982} C_DIS
LIN {X 127.2833,Y 64.0597,Z 181,A 28.5547,B 4.7012,C 0.1802,E1 4.8483,E2 424.4635} C_DIS
LIN {X 128.8148,Y 60.9205,Z 181,A 27.1896,B 4.701,C 0.1832,E1 4.8499,E2 425.824} C_DIS
LIN {X 130.4627,Y 57.3101,Z 181,A 25.5114,B 4.7008,C 0.1885,E1 4.8518,E2 427.5138} C_DIS
LIN {X 132.3026,Y 52.9192,Z 181,A 23.7784,B 4.7008,C 0.1911,E1 4.8537,E2 429.224} C_DIS
LIN {X 133.4597,Y 49.9278,Z 181,A 22.4835,B 4.7006,C 0.1946,E1 4.8549,E2 430.5202} C_DIS
LIN {X 134.743,Y 46.3544,Z 181,A 21.0419,B 4.7005,C 0.1975,E1 4.8563,E2 431.9515} C_DIS
LIN {X 135.8393,Y 43.0361,Z 181,A 19.638,B 4.7003,C 0.2013,E1 4.8575,E2 433.3561} C_DIS
LIN {X 137.085,Y 38.8884,Z 181,A 17.8847,B 4.7001,C 0.2062,E1 4.8589,E2 435.1119} C_DIS
LIN {X 138.1533,Y 34.9001,Z 181,A 16.322,B 4.6999,C 0.2094,E1 4.8599,E2 436.6628} C_DIS
LIN {X 139.2214,Y 30.3617,Z 181,A 14.5118,B 4.6998,C 0.2137,E1 4.8611,E2 438.4657} C_DIS
LIN {X 139.9983,Y 26.5493,Z 181,A 13.0354,B 4.6996,C 0.2168,E1 4.8619,E2 439.9314} C_DIS
LIN {X 140.6856,Y 22.6406,Z 181,A 11.4754,B 4.6994,C 0.2208,E1 4.8626,E2 441.4878} C_DIS
LIN {X 141.1322,Y 19.6551,Z 181,A 10.3144,B 4.6993,C 0.2234,E1 4.863,E2 442.6426} C_DIS
LIN {X 141.5728,Y 16.1864,Z 181,A 8.9543,B 4.6991,C 0.2268,E1 4.8635,E2 443.9977} C_DIS
LIN {X 141.9282,Y 12.6998,Z 181,A 7.5565,B 4.699,C 0.2306,E1 4.8639,E2 445.3949} C_DIS
LIN {X 142.196,Y 9.2151,Z 181,A 6.1132,B 4.6987,C 0.2351,E1 4.8642,E2 446.8442} C_DIS
LIN {X 142.397,Y 5.2526,Z 181,A 4.6716,B 4.6987,C 0.2375,E1 4.8643,E2 448.2666} C_DIS
LIN {X 142.4843,Y 1.745,Z 181,A 3.3046,B 4.6984,C 0.2409,E1 4.8643,E2 449.6289} C_DIS
LIN {X 142.4897,Y -1.1269,Z 181,A 2.1684,B 4.6983,C 0.2439,E1 4.8643,E2 450.7634} C_DIS
LIN {X 142.4159,Y -4.7681,Z 181,A 0.6222,B 4.698,C 0.2492,E1 4.8643,E2 452.3215} C_DIS
LIN {X 142.2549,Y -8.2594,Z 181,A -0.7151,B 4.6978,C 0.2522,E1 4.8641,E2 453.6508} C_DIS
LIN {X 141.9677,Y -12.2318,Z 181,A -2.1622,B 4.6978,C 0.2546,E1 4.8638,E2 455.0787} C_DIS
LIN {X 141.6258,Y -15.7076,Z 181,A -3.5218,B 4.6975,C 0.258,E1 4.8634,E2 456.4334} C_DIS
LIN {X 141.1989,Y -19.1748,Z 181,A -4.8827,B 4.6973,C 0.2613,E1 4.8629,E2 457.7896} C_DIS
LIN {X 140.7599,Y -22.1617,Z 181,A -6.0676,B 4.6972,C 0.2643,E1 4.8624,E2 458.9716} C_DIS
LIN {X 140.0893,Y -26.0734,Z 181,A -7.5614,B 4.697,C 0.2674,E1 4.8617,E2 460.4531} C_DIS
LIN {X 139.4042,Y -29.515,Z 181,A -8.8952,B 4.6968,C 0.2702,E1 4.8609,E2 461.7777} C_DIS
LIN {X 138.6398,Y -32.9176,Z 181,A -10.3567,B 4.6966,C 0.275,E1 4.86,E2 463.2482} C_DIS
LIN {X 137.7925,Y -36.3006,Z 181,A -11.7177,B 4.6964,C 0.2783,E1 4.8591,E2 464.6048} C_DIS
LIN {X 136.9914,Y -39.2222,Z 181,A -12.9007,B 4.6962,C 0.2811,E1 4.8582,E2 465.7843} C_DIS
LIN {X 135.9883,Y -42.5697,Z 181,A -14.2488,B 4.696,C 0.2842,E1 4.8571,E2 467.1259} C_DIS
LIN {X 134.8985,Y -45.9058,Z 181,A -15.6361,B 4.6958,C 0.2877,E1 4.8559,E2 468.5112} C_DIS
LIN {X 133.9997,Y -48.4601,Z 181,A -16.7831,B 4.6956,C 0.2914,E1 4.8548,E2 469.6669} C_DIS
LIN {X 132.4835,Y -52.4704,Z 181,A -18.3661,B 4.6954,C 0.2941,E1 4.8532,E2 471.2325} C_DIS
LIN {X 131.1565,Y -55.7045,Z 181,A -19.7413,B 4.6952,C 0.2974,E1 4.8517,E2 472.6048} C_DIS
LIN {X 129.9134,Y -58.5399,Z 181,A -20.9498,B 4.695,C 0.3001,E1 4.8503,E2 473.8095} C_DIS
LIN {X 128.1635,Y -62.2823,Z 181,A -22.5563,B 4.6948,C 0.3037,E1 4.8484,E2 475.41} C_DIS
LIN {X 126.8883,Y -64.8356,Z 181,A -23.6818,B 4.6946,C 0.3063,E1 4.847,E2 476.5335} C_DIS
LIN {X 125.1408,Y -68.1514,Z 181,A -25.2438,B 4.6943,C 0.3109,E1 4.8449,E2 478.1043} C_DIS
LIN {X 122.9074,Y -72.1015,Z 181,A -26.9989,B 4.6941,C 0.3145,E1 4.8425,E2 479.8517} C_DIS
LIN {X 120.5108,Y -76.0394,Z 181,A -28.7998,B 4.6938,C 0.3184,E1 4.8399,E2 481.6471} C_DIS
LIN {X 117.9946,Y -79.8882,Z 181,A -30.6319,B 4.6935,C 0.3226,E1 4.837,E2 483.4785} C_DIS
LIN {X 115.4947,Y -83.4617,Z 181,A -32.3454,B 4.6933,C 0.3262,E1 4.8343,E2 485.1881} C_DIS
LIN {X 112.884,Y -86.961,Z 181,A -34.0793,B 4.693,C 0.33,E1 4.8313,E2 486.9207} C_DIS
LIN {X 110.1508,Y -90.3976,Z 181,A -35.7101,B 4.6929,C 0.3322,E1 4.8285,E2 488.5347} C_DIS
LIN {X 107.4851,Y -93.5511,Z 181,A -37.3435,B 4.6926,C 0.3355,E1 4.8255,E2 490.1659} C_DIS
LIN {X 104.5673,Y -96.8023,Z 181,A -39.0657,B 4.6924,C 0.3388,E1 4.8223,E2 491.885} C_DIS
LIN {X 101.5424,Y -99.9702,Z 181,A -40.7713,B 4.6922,C 0.3418,E1 4.819,E2 493.5846} C_DIS
LIN {X 98.718,Y -102.7605,Z 181,A -42.4181,B 4.6919,C 0.3458,E1 4.8157,E2 495.2396} C_DIS
LIN {X 95.2264,Y -106.0038,Z 181,A -44.2601,B 4.6917,C 0.3486,E1 4.8119,E2 497.0732} C_DIS
LIN {X 91.7413,Y -109.034,Z 181,A -46.1001,B 4.6914,C 0.3519,E1 4.808,E2 498.9124} C_DIS
LIN {X 88.3574,Y -111.7944,Z 181,A -47.8399,B 4.6912,C 0.355,E1 4.8042,E2 500.6515} C_DIS
LIN {X 84.698,Y -114.5917,Z 181,A -49.616,B 4.691,C 0.3573,E1 4.8003,E2 502.4188} C_DIS
LIN {X 81.1342,Y -117.1417,Z 181,A -51.3805,B 4.6908,C 0.3604,E1 4.7963,E2 504.1851} C_DIS
LIN {X 77.1753,Y -119.7872,Z 181,A -53.1953,B 4.6907,C 0.3623,E1 4.792,E2 505.9878} C_DIS
LIN {X 73.4707,Y -122.0942,Z 181,A -54.9576,B 4.6904,C 0.3652,E1 4.7878,E2 507.7525} C_DIS
LIN {X 69.4894,Y -124.4034,Z 181,A -56.7352,B 4.6903,C 0.367,E1 4.7835,E2 509.5216} C_DIS
LIN {X 65.8668,Y -126.3566,Z 181,A -58.3491,B 4.6901,C 0.3689,E1 4.7796,E2 511.1311} C_DIS
LIN {X 62.4947,Y -128.0587,Z 181,A -59.764,B 4.6901,C 0.3697,E1 4.7761,E2 512.533} C_DIS
LIN {X 59.5517,Y -129.4524,Z 181,A -61.1372,B 4.6899,C 0.3722,E1 4.7726,E2 513.9159} C_DIS
LIN {X 56.161,Y -130.9595,Z 181,A -62.5857,B 4.6898,C 0.3735,E1 4.7689,E2 515.3595} C_DIS
LIN {X 52.9145,Y -132.3045,Z 181,A -63.9781,B 4.6897,C 0.3749,E1 4.7653,E2 516.7501} C_DIS
LIN {X 49.6551,Y -133.5619,Z 181,A -65.3654,B 4.6896,C 0.3763,E1 4.7617,E2 518.136} C_DIS
LIN {X 46.3656,Y -134.7391,Z 181,A -66.7536,B 4.6895,C 0.3776,E1 4.758,E2 519.5229} C_DIS
LIN {X 43.0333,Y -135.8402,Z 181,A -68.1509,B 4.6894,C 0.3788,E1 4.7543,E2 520.9193} C_DIS
LIN {X 39.2273,Y -136.9899,Z 181,A -69.9201,B 4.6891,C 0.3823,E1 4.7495,E2 522.7129} C_DIS
LIN {X 35.0913,Y -138.1048,Z 181,A -71.4391,B 4.6891,C 0.3813,E1 4.7454,E2 524.2052} C_DIS
LIN {X 31.7006,Y -138.9223,Z 181,A -72.8325,B 4.6891,C 0.3823,E1 4.7417,E2 525.5982} C_DIS
LIN {X 28.2688,Y -139.6612,Z 181,A -74.229,B 4.6891,C 0.3831,E1 4.7378,E2 526.9936} C_DIS
LIN {X 24.8373,Y -140.3123,Z 181,A -75.6629,B 4.6889,C 0.3844,E1 4.7339,E2 528.4323} C_DIS
LIN {X 20.9209,Y -140.9513,Z 181,A -77.1764,B 4.6889,C 0.3844,E1 4.7297,E2 529.9356} C_DIS
LIN {X 17.9265,Y -141.3625,Z 181,A -78.4084,B 4.6889,C 0.3851,E1 4.7263,E2 531.1706} C_DIS
LIN {X 14.4416,Y -141.762,Z 181,A -79.8384,B 4.6888,C 0.386,E1 4.7223,E2 532.604} C_DIS
LIN {X 10.9604,Y -142.0726,Z 181,A -81.2379,B 4.6888,C 0.3864,E1 4.7184,E2 534.0034} C_DIS
LIN {X 7.0016,Y -142.3215,Z 181,A -82.8078,B 4.6888,C 0.3866,E1 4.7141,E2 535.5708} C_DIS
LIN {X 3.4957,Y -142.4515,Z 181,A -84.2044,B 4.6888,C 0.3868,E1 4.7102,E2 536.9661} C_DIS
LIN {X 1.0245,Y -142.4893,Z 181,A -84.9136,B 4.689,C 0.3837,E1 4.7083,E2 537.6368} C_DIS
Enddeposition()
LIN {X 0.9671,Y -133.5517,Z 182,A -85.0693,B 4.4546,C 0.3542,E1 4.4724,E2 537.5571} C_DIS
Startdeposition()
$VEL.CP = VEL_PRINT
LIN {X 3.2738,Y -133.5166,Z 182,A -83.6637,B 4.4549,C 0.3498,E1 4.4765,E2 536.0981} C_DIS
LIN {X 6.8422,Y -133.3806,Z 182,A -82.2664,B 4.4549,C 0.3508,E1 4.4803,E2 534.7172} C_DIS
LIN {X 10.0997,Y -133.174,Z 182,A -80.8578,B 4.4549,C 0.3502,E1 4.4842,E2 533.3068} C_DIS
LIN {X 13.0615,Y -132.916,Z 182,A -79.5524,B 4.4549,C 0.3494,E1 4.4879,E2 531.9968} C_DIS
LIN {X 16.347,Y -132.5527,Z 182,A -78.0903,B 4.455,C 0.3483,E1 4.492,E2 530.5284} C_DIS
LIN {X 19.8878,Y -132.0679,Z 182,A -76.6044,B 4.455,C 0.348,E1 4.4961,E2 529.0477} C_DIS
LIN {X 22.8174,Y -131.5941,Z 182,A -75.3389,B 4.4551,C 0.3473,E1 4.4995,E2 527.7824} C_DIS
LIN {X 26.0362,Y -130.9947,Z 182,A -73.8624,B 4.4552,C 0.3456,E1 4.5036,E2 526.2958} C_DIS
LIN {X 29.558,Y -130.2439,Z 182,A -72.5028,B 4.4552,C 0.3464,E1 4.5073,E2 524.9588} C_DIS
LIN {X 32.7421,Y -129.48,Z 182,A -71.0297,B 4.4553,C 0.3446,E1 4.5113,E2 523.4762} C_DIS
LIN {X 35.9081,Y -128.6379,Z 182,A -69.5681,B 4.4555,C 0.3427,E1 4.5153,E2 522.0065} C_DIS
LIN {X 39.7344,Y -127.5097,Z 182,A -67.7916,B 4.4556,C 0.3404,E1 4.52,E2 520.2206} C_DIS
LIN {X 43.4612,Y -126.2866,Z 182,A -66.2844,B 4.4556,C 0.3406,E1 4.524,E2 518.7347} C_DIS
LIN {X 46.5332,Y -125.1872,Z 182,A -64.9023,B 4.4557,C 0.3393,E1 4.5276,E2 517.3538} C_DIS
LIN {X 49.577,Y -124.0134,Z 182,A -63.5228,B 4.4558,C 0.3379,E1 4.5312,E2 515.9759} C_DIS
LIN {X 52.6207,Y -122.753,Z 182,A -62.1279,B 4.456,C 0.3363,E1 4.5348,E2 514.5823} C_DIS
LIN {X 55.6129,Y -121.4269,Z 182,A -60.7455,B 4.456,C 0.3348,E1 4.5383,E2 513.2017} C_DIS
LIN {X 58.8426,Y -119.8944,Z 182,A -59.2337,B 4.4562,C 0.333,E1 4.5421,E2 511.6915} C_DIS
LIN {X 61.8802,Y -118.3551,Z 182,A -57.9675,B 4.4562,C 0.3332,E1 4.5452,E2 510.449} C_DIS
LIN {X 65.0257,Y -116.6593,Z 182,A -56.156,B 4.4566,C 0.3277,E1 4.5497,E2 508.601} C_DIS
LIN {X 68.9301,Y -114.3952,Z 182,A -54.3848,B 4.4566,C 0.3266,E1 4.5539,E2 506.8494} C_DIS
LIN {X 71.716,Y -112.67,Z 182,A -53.0077,B 4.4568,C 0.3247,E1 4.5572,E2 505.4748} C_DIS
LIN {X 74.4557,Y -110.8786,Z 182,A -51.5544,B 4.457,C 0.3218,E1 4.5606,E2 504.0142} C_DIS
LIN {X 77.9856,Y -108.4249,Z 182,A -49.7501,B 4.4572,C 0.3191,E1 4.5647,E2 502.2135} C_DIS
LIN {X 81.0625,Y -106.1436,Z 182,A -48.1086,B 4.4574,C 0.3161,E1 4.5683,E2 500.5708} C_DIS
LIN {X 84.2122,Y -103.6631,Z 182,A -46.3865,B 4.4577,C 0.3129,E1 4.5721,E2 498.847} C_DIS
LIN {X 87.2325,Y -101.134,Z 182,A -44.8394,B 4.4577,C 0.3114,E1 4.5753,E2 497.3168} C_DIS
LIN {X 90.2892,Y -98.4147,Z 182,A -43.1202,B 4.458,C 0.3083,E1 4.5789,E2 495.6006} C_DIS
LIN {X 92.7978,Y -96.053,Z 182,A -41.5947,B 4.4582,C 0.3047,E1 4.582,E2 494.0679} C_DIS
LIN {X 96.0535,Y -92.7972,Z 182,A -39.7493,B 4.4584,C 0.3022,E1 4.5856,E2 492.2373} C_DIS
LIN {X 98.5036,Y -90.1925,Z 182,A -38.1491,B 4.4587,C 0.2981,E1 4.5886,E2 490.6274} C_DIS
LIN {X 101.5528,Y -86.7451,Z 182,A -36.3141,B 4.4588,C 0.2954,E1 4.592,E2 488.8085} C_DIS
LIN {X 104.1775,Y -83.5749,Z 182,A -34.6075,B 4.4591,C 0.2922,E1 4.595,E2 487.1079} C_DIS
LIN {X 106.5474,Y -80.531,Z 182,A -33.0527,B 4.4592,C 0.2896,E1 4.5976,E2 485.5643} C_DIS
LIN {X 108.4127,Y -78.0028,Z 182,A -31.7019,B 4.4594,C 0.2864,E1 4.5998,E2 484.212} C_DIS
LIN {X 110.1323,Y -75.5544,Z 182,A -30.4556,B 4.4596,C 0.2838,E1 4.6018,E2 482.9693} C_DIS
LIN {X 111.952,Y -72.831,Z 182,A -29.0906,B 4.4598,C 0.2809,E1 4.6039,E2 481.6081} C_DIS
LIN {X 113.7039,Y -70.0648,Z 182,A -27.7257,B 4.46,C 0.278,E1 4.6059,E2 480.2471} C_DIS
LIN {X 115.5384,Y -66.9961,Z 182,A -26.2285,B 4.4602,C 0.2746,E1 4.608,E2 478.7532} C_DIS
LIN {X 117.1658,Y -64.1077,Z 182,A -24.8306,B 4.4604,C 0.2713,E1 4.6099,E2 477.3572} C_DIS
LIN {X 118.5574,Y -61.4951,Z 182,A -23.606,B 4.4605,C 0.2687,E1 4.6115,E2 476.1372} C_DIS
LIN {X 120.0276,Y -58.5725,Z 182,A -22.2282,B 4.4607,C 0.2654,E1 4.6132,E2 474.7614} C_DIS
LIN {X 121.5551,Y -55.3356,Z 182,A -20.7523,B 4.4609,C 0.2621,E1 4.6149,E2 473.2917} C_DIS
LIN {X 122.8736,Y -52.3416,Z 182,A -19.3915,B 4.4611,C 0.259,E1 4.6164,E2 471.9351} C_DIS
LIN {X 124.1187,Y -49.3159,Z 182,A -18.028,B 4.4613,C 0.2557,E1 4.6179,E2 470.5755} C_DIS
LIN {X 125.2936,Y -46.2493,Z 182,A -16.6808,B 4.4615,C 0.2527,E1 4.6192,E2 469.2348} C_DIS
LIN {X 126.3865,Y -43.173,Z 182,A -15.3079,B 4.4617,C 0.2493,E1 4.6204,E2 467.8642} C_DIS
LIN {X 127.5449,Y -39.6196,Z 182,A -13.6172,B 4.462,C 0.2438,E1 4.6219,E2 466.1612} C_DIS
LIN {X 128.7202,Y -35.6138,Z 182,A -12.0179,B 4.462,C 0.2414,E1 4.6231,E2 464.5845} C_DIS
LIN {X 129.6298,Y -32.1519,Z 182,A -10.539,B 4.4623,C 0.2378,E1 4.6241,E2 463.1115} C_DIS
LIN {X 130.312,Y -29.2599,Z 182,A -9.2664,B 4.4625,C 0.2343,E1 4.6249,E2 461.8381} C_DIS
LIN {X 131.0502,Y -25.7576,Z 182,A -7.7943,B 4.4626,C 0.2308,E1 4.6257,E2 460.3727} C_DIS
LIN {X 131.5903,Y -22.839,Z 182,A -6.58,B 4.4628,C 0.228,E1 4.6263,E2 459.1649} C_DIS
LIN {X 132.1129,Y -19.5913,Z 182,A -5.1084,B 4.463,C 0.2233,E1 4.6269,E2 457.6846} C_DIS
LIN {X 132.5886,Y -16.0461,Z 182,A -3.7113,B 4.4632,C 0.2207,E1 4.6274,E2 456.3034} C_DIS
LIN {X 132.9418,Y -12.7922,Z 182,A -2.4177,B 4.4632,C 0.2182,E1 4.6278,E2 455.0225} C_DIS
LIN {X 133.2155,Y -9.5312,Z 182,A -1.0454,B 4.4635,C 0.2146,E1 4.6281,E2 453.6531} C_DIS
LIN {X 133.4268,Y -5.9142,Z 182,A 0.4713,B 4.4636,C 0.2107,E1 4.6283,E2 452.14} C_DIS
LIN {X 133.5249,Y -2.9723,Z 182,A 1.7542,B 4.4638,C 0.2068,E1 4.6283,E2 450.8536} C_DIS
LIN {X 133.5563,Y 0.4744,Z 182,A 3.073,B 4.4639,C 0.2047,E1 4.6284,E2 449.5536} C_DIS
LIN {X 133.5168,Y 3.2663,Z 182,A 4.4018,B 4.4642,C 0.1996,E1 4.6284,E2 448.2077} C_DIS
LIN {X 133.3795,Y 6.865,Z 182,A 5.7718,B 4.4642,C 0.1975,E1 4.6282,E2 446.8582} C_DIS
LIN {X 133.1717,Y 10.1309,Z 182,A 7.1453,B 4.4644,C 0.1939,E1 4.6279,E2 445.4876} C_DIS
LIN {X 132.9134,Y 13.0884,Z 182,A 8.4097,B 4.4646,C 0.1904,E1 4.6276,E2 444.2235} C_DIS
LIN {X 132.5534,Y 16.3411,Z 182,A 9.8221,B 4.4647,C 0.1863,E1 4.6271,E2 442.8092} C_DIS
LIN {X 132.0653,Y 19.9042,Z 182,A 11.282,B 4.4649,C 0.1831,E1 4.6265,E2 441.3585} C_DIS
LIN {X 131.591,Y 22.835,Z 182,A 12.5175,B 4.4649,C 0.18,E1 4.626,E2 440.1269} C_DIS
LIN {X 130.9908,Y 26.0555,Z 182,A 13.9537,B 4.4652,C 0.1757,E1 4.6252,E2 438.686} C_DIS
LIN {X 130.245,Y 29.5533,Z 182,A 15.278,B 4.4652,C 0.1741,E1 4.6244,E2 437.3866} C_DIS
LIN {X 129.4775,Y 32.752,Z 182,A 16.7264,B 4.4654,C 0.1697,E1 4.6234,E2 435.9329} C_DIS
LIN {X 128.6353,Y 35.9174,Z 182,A 18.0889,B 4.4655,C 0.1664,E1 4.6224,E2 434.5748} C_DIS
LIN {X 127.7159,Y 39.0606,Z 182,A 19.3809,B 4.4655,C 0.164,E1 4.6214,E2 433.2959} C_DIS
LIN {X 126.7417,Y 42.1145,Z 182,A 20.799,B 4.4658,C 0.1598,E1 4.6202,E2 431.8718} C_DIS
LIN {X 125.7558,Y 44.9742,Z 182,A 22.0387,B 4.4658,C 0.157,E1 4.619,E2 430.6385} C_DIS
LIN {X 124.6331,Y 47.9982,Z 182,A 23.3709,B 4.466,C 0.154,E1 4.6177,E2 429.312} C_DIS
LIN {X 123.489,Y 50.8719,Z 182,A 24.7491,B 4.466,C 0.1499,E1 4.6163,E2 427.9269} C_DIS
LIN {X 122.0974,Y 54.1247,Z 182,A 26.1463,B 4.4662,C 0.1474,E1 4.6147,E2 426.5437} C_DIS
LIN {X 120.7347,Y 57.1003,Z 182,A 27.5901,B 4.4663,C 0.1433,E1 4.613,E2 425.0944} C_DIS
LIN {X 119.0571,Y 60.5182,Z 182,A 28.9352,B 4.4663,C 0.1427,E1 4.6114,E2 423.7837} C_DIS
LIN {X 117.7863,Y 62.9607,Z 182,A 30.3248,B 4.4665,C 0.1372,E1 4.6095,E2 422.3684} C_DIS
LIN {X 116.2015,Y 65.8403,Z 182,A 31.69,B 4.4665,C 0.1342,E1 4.6077,E2 421.0081} C_DIS
LIN {X 114.3958,Y 68.9292,Z 182,A 33.111,B 4.4667,C 0.1319,E1 4.6057,E2 419.6004} C_DIS
LIN {X 112.6729,Y 71.7114,Z 182,A 34.4743,B 4.4667,C 0.129,E1 4.6037,E2 418.2415} C_DIS
LIN {X 110.8822,Y 74.4503,Z 182,A 35.8086,B 4.4668,C 0.1265,E1 4.6016,E2 416.9151} C_DIS
LIN {X 108.9021,Y 77.3181,Z 182,A 37.2309,B 4.4668,C 0.1238,E1 4.5994,E2 415.5012} C_DIS
LIN {X 107.042,Y 79.8725,Z 182,A 38.7322,B 4.467,C 0.119,E1 4.5968,E2 413.9818} C_DIS
LIN {X 104.2727,Y 83.4561,Z 182,A 40.5743,B 4.4671,C 0.1158,E1 4.5937,E2 412.1514} C_DIS
LIN {X 101.5715,Y 86.7231,Z 182,A 42.3964,B 4.4672,C 0.1118,E1 4.5904,E2 410.3284} C_DIS
LIN {X 98.9601,Y 89.6911,Z 182,A 43.9776,B 4.4672,C 0.1095,E1 4.5875,E2 408.7608} C_DIS
LIN {X 96.1659,Y 92.6811,Z 182,A 45.7907,B 4.4674,C 0.1052,E1 4.584,E2 406.9403} C_DIS
LIN {X 93.276,Y 95.5892,Z 182,A 47.5153,B 4.4674,C 0.102,E1 4.5806,E2 405.2195} C_DIS
LIN {X 90.1972,Y 98.4993,Z 182,A 49.2892,B 4.4675,C 0.099,E1 4.5769,E2 403.4506} C_DIS
LIN {X 86.7305,Y 101.5652,Z 182,A 51.136,B 4.4675,C 0.0968,E1 4.5731,E2 401.6203} C_DIS
LIN {X 83.5728,Y 104.1792,Z 182,A 52.849,B 4.4676,C 0.0941,E1 4.5694,E2 399.9126} C_DIS
LIN {X 80.6355,Y 106.4686,Z 182,A 54.4919,B 4.4676,C 0.0908,E1 4.5657,E2 398.2641} C_DIS
LIN {X 77.9922,Y 108.4202,Z 182,A 55.8686,B 4.4677,C 0.0888,E1 4.5626,E2 396.8913} C_DIS
LIN {X 74.4486,Y 110.8833,Z 182,A 57.6599,B 4.4677,C 0.0864,E1 4.5585,E2 395.1072} C_DIS
LIN {X 71.4517,Y 112.8374,Z 182,A 59.0957,B 4.4677,C 0.0851,E1 4.5552,E2 393.6832} C_DIS
LIN {X 68.6666,Y 114.5539,Z 182,A 60.5463,B 4.4678,C 0.0825,E1 4.5517,E2 392.227} C_DIS
LIN {X 65.5756,Y 116.3506,Z 182,A 62.02,B 4.4678,C 0.0809,E1 4.5481,E2 390.7605} C_DIS
LIN {X 62.6901,Y 117.9298,Z 182,A 63.5035,B 4.4679,C 0.0781,E1 4.5445,E2 389.2685} C_DIS
LIN {X 59.1943,Y 119.7209,Z 182,A 65.1065,B 4.4679,C 0.0768,E1 4.5405,E2 387.6753} C_DIS
LIN {X 55.3375,Y 121.5542,Z 182,A 66.8494,B 4.4679,C 0.0755,E1 4.5361,E2 385.9434} C_DIS
LIN {X 51.9833,Y 123.0248,Z 182,A 68.2949,B 4.4679,C 0.075,E1 4.5324,E2 384.5131} C_DIS
LIN {X 49.3163,Y 124.1185,Z 182,A 69.6177,B 4.468,C 0.0727,E1 4.529,E2 383.1802} C_DIS
LIN {X 46.2605,Y 125.2894,Z 182,A 70.9862,B 4.468,C 0.0716,E1 4.5254,E2 381.8161} C_DIS
LIN {X 43.1208,Y 126.4046,Z 182,A 72.4909,B 4.468,C 0.0694,E1 4.5214,E2 380.3026} C_DIS
LIN {X 38.8347,Y 127.7851,Z 182,A 74.3181,B 4.468,C 0.0687,E1 4.5166,E2 378.4883} C_DIS
LIN {X 35.1437,Y 128.8511,Z 182,A 75.9364,B 4.468,C 0.0676,E1 4.5122,E2 376.8741} C_DIS
LIN {X 32.1566,Y 129.6286,Z 182,A 77.263,B 4.4681,C 0.0666,E1 4.5086,E2 375.5475} C_DIS
LIN {X 29.2649,Y 130.3109,Z 182,A 78.5607,B 4.4681,C 0.0655,E1 4.5051,E2 374.2474} C_DIS
LIN {X 25.6019,Y 131.08,Z 182,A 80.0889,B 4.4681,C 0.0652,E1 4.5009,E2 372.7288} C_DIS
LIN {X 22.8331,Y 131.5913,Z 182,A 81.3199,B 4.4681,C 0.0643,E1 4.4975,E2 371.4955} C_DIS
LIN {X 19.601,Y 132.1116,Z 182,A 82.8254,B 4.4681,C 0.0627,E1 4.4934,E2 369.9784} C_DIS
LIN {X 16.0528,Y 132.5878,Z 182,A 84.2599,B 4.4681,C 0.063,E1 4.4894,E2 368.5564} C_DIS
LIN {X 12.7983,Y 132.9412,Z 182,A 85.6505,B 4.4681,C 0.0626,E1 4.4856,E2 367.1679} C_DIS
LIN {X 9.521,Y 133.2163,Z 182,A 87.009,B 4.4681,C 0.0627,E1 4.4818,E2 365.8162} C_DIS
LIN {X 5.9542,Y 133.4253,Z 182,A 88.5645,B 4.4681,C 0.0622,E1 4.4774,E2 364.2586} C_DIS
LIN {X 2.9877,Y 133.5245,Z 182,A 89.8781,B 4.4681,C 0.0616,E1 4.4738,E2 362.9408} C_DIS
LIN {X 0.0159,Y 133.558,Z 182,A 91.1559,B 4.4681,C 0.0616,E1 4.4702,E2 361.6633} C_DIS
LIN {X -3.28,Y 133.5164,Z 182,A 92.6267,B 4.4681,C 0.061,E1 4.4661,E2 360.1863} C_DIS
LIN {X -6.8533,Y 133.3801,Z 182,A 94.0547,B 4.4681,C 0.062,E1 4.4621,E2 358.7716} C_DIS
LIN {X -10.117,Y 133.1728,Z 182,A 95.4494,B 4.4681,C 0.0623,E1 4.4582,E2 357.3786} C_DIS
LIN {X -13.0765,Y 132.9145,Z 182,A 96.7592,B 4.4681,C 0.0623,E1 4.4546,E2 356.0651} C_DIS
LIN {X -16.3509,Y 132.5522,Z 182,A 98.2346,B 4.4681,C 0.062,E1 4.4505,E2 354.5832} C_DIS
LIN {X -19.8974,Y 132.0664,Z 182,A 99.7353,B 4.4681,C 0.0629,E1 4.4463,E2 353.0874} C_DIS
LIN {X -22.8264,Y 131.5925,Z 182,A 101.035,B 4.4681,C 0.0632,E1 4.4427,E2 351.7853} C_DIS
LIN {X -26.0449,Y 130.9929,Z 182,A 102.5063,B 4.4681,C 0.0632,E1 4.4387,E2 350.3067} C_DIS
LIN {X -29.943,Y 130.156,Z 182,A 104.2226,B 4.4681,C 0.0641,E1 4.434,E2 348.5907} C_DIS
LIN {X -34.3325,Y 129.0674,Z 182,A 106.0944,B 4.4681,C 0.066,E1 4.429,E2 346.7281} C_DIS
LIN {X -37.4868,Y 128.1867,Z 182,A 107.5932,B 4.4681,C 0.0662,E1 4.4249,E2 345.2191} C_DIS
LIN {X -42.0048,Y 126.7782,Z 182,A 109.6227,B 4.4681,C 0.0678,E1 4.4195,E2 343.1909} C_DIS
LIN {X -44.978,Y 125.7544,Z 182,A 110.9197,B 4.4681,C 0.0694,E1 4.4161,E2 341.901} C_DIS
LIN {X -48.0293,Y 124.621,Z 182,A 112.3442,B 4.4681,C 0.0705,E1 4.4124,E2 340.4741} C_DIS
LIN {X -51.1058,Y 123.3913,Z 182,A 113.7699,B 4.4681,C 0.0719,E1 4.4087,E2 339.0488} C_DIS
LIN {X -54.1234,Y 122.0979,Z 182,A 115.1958,B 4.4681,C 0.0733,E1 4.405,E2 337.6219} C_DIS
LIN {X -57.1008,Y 120.7345,Z 182,A 116.7022,B 4.468,C 0.0741,E1 4.4012,E2 336.1043} C_DIS
LIN {X -60.3142,Y 119.161,Z 182,A 118.0704,B 4.468,C 0.0773,E1 4.3978,E2 334.7569} C_DIS
LIN {X -62.9487,Y 117.7928,Z 182,A 119.5493,B 4.468,C 0.0773,E1 4.3941,E2 333.2546} C_DIS
LIN {X -65.8375,Y 116.2031,Z 182,A 120.9788,B 4.468,C 0.0791,E1 4.3906,E2 331.8244} C_DIS
LIN {X -68.9116,Y 114.4064,Z 182,A 122.4537,B 4.4679,C 0.0816,E1 4.3871,E2 330.3568} C_DIS
LIN {X -71.6768,Y 112.6951,Z 182,A 123.8794,B 4.4679,C 0.0835,E1 4.3837,E2 328.9286} C_DIS
LIN {X -74.3932,Y 110.9203,Z 182,A 125.2502,B 4.4678,C 0.0857,E1 4.3805,E2 327.5613} C_DIS
LIN {X -76.8293,Y 109.2469,Z 182,A 126.6622,B 4.4678,C 0.0866,E1 4.3773,E2 326.1331} C_DIS
LIN {X -79.5676,Y 107.269,Z 182,A 128.0978,B 4.4678,C 0.0891,E1 4.374,E2 324.7002} C_DIS
LIN {X -82.8167,Y 104.7814,Z 182,A 129.8865,B 4.4677,C 0.0919,E1 4.3701,E2 322.9089} C_DIS
LIN {X -85.9884,Y 102.194,Z 182,A 131.651,B 4.4676,C 0.0949,E1 4.3663,E2 321.1448} C_DIS
LIN {X -88.9522,Y 99.6249,Z 182,A 133.4347,B 4.4676,C 0.0973,E1 4.3625,E2 319.3504} C_DIS
LIN {X -92.0969,Y 96.7254,Z 182,A 135.2761,B 4.4675,C 0.1007,E1 4.3588,E2 317.5096} C_DIS
LIN {X -95.0189,Y 93.8571,Z 182,A 137.1832,B 4.4675,C 0.1031,E1 4.355,E2 315.5859} C_DIS
LIN {X -97.8493,Y 90.9017,Z 182,A 138.885,B 4.4673,C 0.1071,E1 4.3517,E2 313.892} C_DIS
LIN {X -100.6887,Y 87.7461,Z 182,A 140.7076,B 4.4673,C 0.1109,E1 4.3484,E2 312.0707} C_DIS
LIN {X -103.2424,Y 84.727,Z 182,A 142.5733,B 4.4672,C 0.1134,E1 4.345,E2 310.1861} C_DIS
LIN {X -105.7914,Y 81.5224,Z 182,A 144.1609,B 4.467,C 0.1184,E1 4.3423,E2 308.6202} C_DIS
LIN {X -107.454,Y 79.3178,Z 182,A 145.4555,B 4.467,C 0.1203,E1 4.3401,E2 307.3134} C_DIS
LIN {X -109.7126,Y 76.1626,Z 182,A 147.3258,B 4.467,C 0.1228,E1 4.3371,E2 305.4197} C_DIS
LIN {X -111.9663,Y 72.8089,Z 182,A 148.9504,B 4.4668,C 0.1276,E1 4.3346,E2 303.8096} C_DIS
LIN {X -113.7141,Y 70.0482,Z 182,A 150.3899,B 4.4667,C 0.1307,E1 4.3324,E2 302.3668} C_DIS
LIN {X -115.7546,Y 66.6226,Z 182,A 152.0878,B 4.4666,C 0.1349,E1 4.33,E2 300.6719} C_DIS
LIN {X -117.1516,Y 64.1336,Z 182,A 153.4301,B 4.4666,C 0.1372,E1 4.3282,E2 299.3164} C_DIS
LIN {X -118.5467,Y 61.5154,Z 182,A 154.733,B 4.4664,C 0.1402,E1 4.3265,E2 298.0109} C_DIS
LIN {X -120.301,Y 58.0081,Z 182,A 156.326,B 4.4663,C 0.145,E1 4.3246,E2 296.43} C_DIS
LIN {X -121.5557,Y 55.3343,Z 182,A 157.7709,B 4.4662,C 0.1471,E1 4.3228,E2 294.9648} C_DIS
LIN {X -123.1061,Y 51.7886,Z 182,A 159.2888,B 4.466,C 0.1524,E1 4.3212,E2 293.4653} C_DIS
LIN {X -124.1232,Y 49.3046,Z 182,A 160.6663,B 4.466,C 0.1539,E1 4.3197,E2 292.0615} C_DIS
LIN {X -125.3003,Y 46.2314,Z 182,A 162.1051,B 4.4658,C 0.1575,E1 4.3183,E2 290.6206} C_DIS
LIN {X -126.3941,Y 43.151,Z 182,A 163.566,B 4.4658,C 0.1609,E1 4.317,E2 289.1538} C_DIS
LIN {X -127.4823,Y 39.824,Z 182,A 165.3219,B 4.4656,C 0.1633,E1 4.3155,E2 287.3683} C_DIS
LIN {X -128.7162,Y 35.6281,Z 182,A 167.0504,B 4.4654,C 0.1693,E1 4.3141,E2 285.6591} C_DIS
LIN {X -129.6232,Y 32.1779,Z 182,A 168.6209,B 4.4652,C 0.1733,E1 4.3131,E2 284.0851} C_DIS
LIN {X -130.307,Y 29.2819,Z 182,A 169.9867,B 4.4652,C 0.1763,E1 4.3122,E2 282.7094} C_DIS
LIN {X -131.0529,Y 25.7434,Z 182,A 171.5625,B 4.465,C 0.1804,E1 4.3113,E2 281.1319} C_DIS
LIN {X -131.5928,Y 22.8249,Z 182,A 172.8576,B 4.4648,C 0.1838,E1 4.3107,E2 279.8352} C_DIS
LIN {X -132.1125,Y 19.5941,Z 182,A 174.4219,B 4.4648,C 0.1867,E1 4.31,E2 278.2523} C_DIS
LIN {X -132.5887,Y 16.0452,Z 182,A 175.9117,B 4.4645,C 0.1914,E1 4.3095,E2 276.7693} C_DIS
LIN {X -132.9421,Y 12.7889,Z 182,A 177.2948,B 4.4643,C 0.1955,E1 4.3091,E2 275.3899} C_DIS
LIN {X -133.2169,Y 9.5123,Z 182,A 178.7638,B 4.4642,C 0.1991,E1 4.3088,E2 273.9149} C_DIS
LIN {X -133.3953,Y 6.5508,Z 182,A -179.8397,B 4.464,C 0.2019,E1 4.3086,E2 272.5042} C_DIS
LIN {X -133.5249,Y 2.9739,Z 182,A -178.1643,B 4.4639,C 0.2054,E1 4.3084,E2 270.8128} C_DIS
LIN {X -133.5563,Y -0.4786,Z 182,A -176.8487,B 4.4636,C 0.2106,E1 4.3084,E2 269.5185} C_DIS
LIN {X -133.5163,Y -3.2845,Z 182,A -175.4241,B 4.4636,C 0.2126,E1 4.3084,E2 268.0677} C_DIS
LIN {X -133.3797,Y -6.8607,Z 182,A -173.9724,B 4.4633,C 0.2175,E1 4.3087,E2 266.6273} C_DIS
LIN {X -133.1717,Y -10.1314,Z 182,A -172.5051,B 4.4631,C 0.2211,E1 4.309,E2 265.1534} C_DIS
LIN {X -132.9134,Y -13.0884,Z 182,A -171.1559,B 4.463,C 0.2242,E1 4.3093,E2 263.7958} C_DIS
LIN {X -132.4727,Y -16.9789,Z 182,A -169.5098,B 4.4627,C 0.2291,E1 4.3099,E2 262.1549} C_DIS
LIN {X -132.0655,Y -19.9032,Z 182,A -168.0933,B 4.4627,C 0.2317,E1 4.3104,E2 260.7208} C_DIS
LIN {X -131.5909,Y -22.8357,Z 182,A -166.7766,B 4.4624,C 0.2349,E1 4.311,E2 259.3996} C_DIS
LIN {X -130.9909,Y -26.0547,Z 182,A -165.2433,B 4.4623,C 0.238,E1 4.3119,E2 257.8514} C_DIS
LIN {X -130.2424,Y -29.5648,Z 182,A -163.8302,B 4.462,C 0.2431,E1 4.3127,E2 256.4547} C_DIS
LIN {X -129.4737,Y -32.767,Z 182,A -162.2863,B 4.4618,C 0.2461,E1 4.3137,E2 254.8955} C_DIS
LIN {X -128.6328,Y -35.9264,Z 182,A -160.8386,B 4.4616,C 0.2496,E1 4.3148,E2 253.443} C_DIS
LIN {X -127.7144,Y -39.0655,Z 182,A -159.4661,B 4.4614,C 0.2536,E1 4.3159,E2 252.075} C_DIS
LIN {X -126.8154,Y -41.8933,Z 182,A -158.0072,B 4.4613,C 0.2557,E1 4.3172,E2 250.5938} C_DIS
LIN {X -125.7509,Y -44.9878,Z 182,A -156.6306,B 4.4611,C 0.2596,E1 4.3185,E2 249.2213} C_DIS
LIN {X -124.6112,Y -48.0546,Z 182,A -155.1793,B 4.4609,C 0.263,E1 4.3199,E2 247.7648} C_DIS
LIN {X -123.3891,Y -51.111,Z 182,A -153.7292,B 4.4607,C 0.2664,E1 4.3214,E2 246.3107} C_DIS
LIN {X -122.0979,Y -54.1234,Z 182,A -152.2824,B 4.4605,C 0.2697,E1 4.3231,E2 244.8595} C_DIS
LIN {X -120.735,Y -57.0997,Z 182,A -150.7333,B 4.4603,C 0.2723,E1 4.3249,E2 243.293} C_DIS
LIN {X -119.1585,Y -60.3191,Z 182,A -149.3623,B 4.46,C 0.2773,E1 4.3266,E2 241.9435} C_DIS
LIN {X -117.8002,Y -62.9349,Z 182,A -147.9565,B 4.4599,C 0.2794,E1 4.3284,E2 240.5207} C_DIS
LIN {X -116.24,Y -65.7723,Z 182,A -146.4616,B 4.4597,C 0.2821,E1 4.3305,E2 239.0131} C_DIS
LIN {X -114.2381,Y -69.19,Z 182,A -144.8416,B 4.4594,C 0.2867,E1 4.3328,E2 237.4037} C_DIS
LIN {X -112.6732,Y -71.711,Z 182,A -143.4694,B 4.4593,C 0.289,E1 4.3348,E2 236.0195} C_DIS
LIN {X -110.8832,Y -74.4488,Z 182,A -142.0621,B 4.4591,C 0.2922,E1 4.337,E2 234.6121} C_DIS
LIN {X -109.199,Y -76.8972,Z 182,A -140.7117,B 4.4589,C 0.2946,E1 4.3392,E2 233.2527} C_DIS
LIN {X -107.2719,Y -79.5637,Z 182,A -139.2311,B 4.4587,C 0.2972,E1 4.3416,E2 231.7638} C_DIS
LIN {X -104.7849,Y -82.8122,Z 182,A -137.4341,B 4.4585,C 0.3007,E1 4.3447,E2 229.9621} C_DIS
LIN {X -102.1936,Y -85.9888,Z 182,A -135.6581,B 4.4583,C 0.3043,E1 4.3479,E2 228.1844} C_DIS
LIN {X -99.9526,Y -88.5837,Z 182,A -134.0562,B 4.4581,C 0.3064,E1 4.3509,E2 226.5664} C_DIS
LIN {X -97.1854,Y -91.6111,Z 182,A -132.2338,B 4.4579,C 0.3094,E1 4.3544,E2 224.7363} C_DIS
LIN {X -94.335,Y -94.544,Z 182,A -130.4298,B 4.4577,C 0.3124,E1 4.3579,E2 222.9265} C_DIS
LIN {X -91.0204,Y -97.7387,Z 182,A -128.4866,B 4.4574,C 0.3164,E1 4.3618,E2 220.9876} C_DIS
LIN {X -88.3571,Y -100.153,Z 182,A -126.8354,B 4.4573,C 0.3183,E1 4.3653,E2 219.3229} C_DIS
LIN {X -84.8472,Y -103.1442,Z 182,A -124.913,B 4.457,C 0.3222,E1 4.3694,E2 217.4077} C_DIS
LIN {X -81.6489,Y -105.6934,Z 182,A -123.2248,B 4.4567,C 0.3256,E1 4.3731,E2 215.728} C_DIS
LIN {X -79.3071,Y -107.4619,Z 182,A -121.8824,B 4.4567,C 0.327,E1 4.3761,E2 214.3752} C_DIS
LIN {X -76.6479,Y -109.3748,Z 182,A -120.4817,B 4.4565,C 0.3292,E1 4.3793,E2 212.9752} C_DIS
LIN {X -74.1984,Y -111.0504,Z 182,A -119.1525,B 4.4564,C 0.3306,E1 4.3824,E2 211.6389} C_DIS
LIN {X -71.456,Y -112.8347,Z 182,A -117.7274,B 4.4562,C 0.3324,E1 4.3858,E2 210.211} C_DIS
LIN {X -68.6674,Y -114.5534,Z 182,A -116.2282,B 4.4562,C 0.3336,E1 4.3894,E2 208.6998} C_DIS
LIN {X -65.576,Y -116.3503,Z 182,A -114.6415,B 4.456,C 0.3351,E1 4.3932,E2 207.1064} C_DIS
LIN {X -61.5023,Y -118.5536,Z 182,A -112.7168,B 4.4558,C 0.338,E1 4.398,E2 205.1894} C_DIS
LIN {X -58.5779,Y -120.025,Z 182,A -111.2786,B 4.4558,C 0.3394,E1 4.4016,E2 203.7468} C_DIS
LIN {X -55.3421,Y -121.5521,Z 182,A -109.7408,B 4.4556,C 0.341,E1 4.4055,E2 202.2085} C_DIS
LIN {X -52.3469,Y -122.8713,Z 182,A -108.3223,B 4.4556,C 0.3423,E1 4.4091,E2 200.7879} C_DIS
LIN {X -49.3204,Y -124.1169,Z 182,A -106.9044,B 4.4554,C 0.3435,E1 4.4128,E2 199.368} C_DIS
LIN {X -46.2102,Y -125.3082,Z 182,A -105.3432,B 4.4554,C 0.3435,E1 4.4169,E2 197.7897} C_DIS
LIN {X -43.2026,Y -126.3762,Z 182,A -104.0852,B 4.4552,C 0.3456,E1 4.4202,E2 196.5455} C_DIS
LIN {X -40.4358,Y -127.2874,Z 182,A -102.7314,B 4.4552,C 0.3456,E1 4.4239,E2 195.1782} C_DIS
LIN {X -35.9164,Y -128.6356,Z 182,A -100.7194,B 4.4552,C 0.3471,E1 4.4293,E2 193.1671} C_DIS
LIN {X -32.1595,Y -129.6279,Z 182,A -99.118,B 4.455,C 0.3486,E1 4.4336,E2 191.5738} C_DIS
LIN {X -29.2584,Y -130.3124,Z 182,A -97.7914,B 4.455,C 0.3488,E1 4.4372,E2 190.2406} C_DIS
LIN {X -25.7568,Y -131.0504,Z 182,A -96.2669,B 4.455,C 0.3496,E1 4.4414,E2 188.717} C_DIS
LIN {X -22.3367,Y -131.6751,Z 182,A -94.9527,B 4.4548,C 0.3518,E1 4.4449,E2 187.4249} C_DIS
LIN {X -19.6056,Y -132.1109,Z 182,A -93.4899,B 4.4549,C 0.3495,E1 4.4491,E2 185.9265} C_DIS
LIN {X -16.0602,Y -132.5869,Z 182,A -91.9581,B 4.4549,C 0.3499,E1 4.4533,E2 184.3944} C_DIS
LIN {X -12.7868,Y -132.9423,Z 182,A -90.6995,B 4.4548,C 0.3516,E1 4.4568,E2 183.1548} C_DIS
LIN {X -9.5271,Y -133.2158,Z 182,A -89.282,B 4.4548,C 0.3516,E1 4.4607,E2 181.735} C_DIS
LIN {X -6.5628,Y -133.3947,Z 182,A -87.9295,B 4.4548,C 0.3508,E1 4.4645,E2 180.372} C_DIS
LIN {X -2.9972,Y -133.5243,Z 182,A -86.4128,B 4.4548,C 0.3508,E1 4.4688,E2 178.8564} C_DIS
LIN {X 0.0056,Y -133.558,Z 182,A -85.1153,B 4.4548,C 0.3506,E1 4.4724,E2 177.5571} C_DIS
LIN {X 0.0056,Y -133.558,Z 182,A -85.1153,B 4.4548,C 0.3506,E1 4.4724,E2 177.5571} C_DIS
Enddeposition()
LIN {X 0.9641,Y -134.4524,Z 182,A -85.5468,B 4.4541,C 0.3615,E1 4.4709,E2 178.1275} C_DIS
Startdeposition()
$VEL.CP = VEL_PRINT
LIN {X -4.1297,Y -134.3946,Z 182,A -87.4624,B 4.4543,C 0.3591,E1 4.4657,E2 180.0117} C_DIS
LIN {X -7.0433,Y -134.2731,Z 182,A -88.6851,B 4.4543,C 0.3589,E1 4.4622,E2 181.2324} C_DIS
LIN {X -10.4409,Y -134.053,Z 182,A -90.162,B 4.4543,C 0.3591,E1 4.4581,E2 182.7132} C_DIS
LIN {X -13.585,Y -133.7713,Z 182,A -91.8532,B 4.454,C 0.3623,E1 4.4533,E2 184.449} C_DIS
LIN {X -16.8432,Y -133.3997,Z 182,A -92.8635,B 4.4544,C 0.3583,E1 4.4506,E2 185.4107} C_DIS
LIN {X -19.3849,Y -133.0531,Z 182,A -94.0155,B 4.4544,C 0.3585,E1 4.4474,E2 186.5705} C_DIS
LIN {X -22.2205,Y -132.6085,Z 182,A -95.2545,B 4.4544,C 0.3583,E1 4.444,E2 187.8119} C_DIS
LIN {X -25.918,Y -131.9373,Z 182,A -96.8501,B 4.4544,C 0.3576,E1 4.4396,E2 189.4074} C_DIS
LIN {X -28.3065,Y -131.4438,Z 182,A -97.9386,B 4.4544,C 0.3576,E1 4.4366,E2 190.5023} C_DIS
LIN {X -31.6231,Y -130.6855,Z 182,A -99.4236,B 4.4544,C 0.3572,E1 4.4326,E2 191.9922} C_DIS
LIN {X -35.8377,Y -129.5937,Z 182,A -101.2812,B 4.4545,C 0.3561,E1 4.4275,E2 193.8507} C_DIS
LIN {X -39.2581,Y -128.5982,Z 182,A -103.2992,B 4.4543,C 0.3595,E1 4.422,E2 195.9323} C_DIS
LIN {X -43.5065,Y -127.2245,Z 182,A -104.5711,B 4.4548,C 0.3524,E1 4.4188,E2 197.1248} C_DIS
LIN {X -46.338,Y -126.2223,Z 182,A -106.2172,B 4.4547,C 0.3546,E1 4.4144,E2 198.8176} C_DIS
LIN {X -51.0189,Y -124.4041,Z 182,A -108.1462,B 4.455,C 0.3508,E1 4.4094,E2 200.7203} C_DIS
LIN {X -53.4662,Y -123.3695,Z 182,A -109.3587,B 4.455,C 0.3503,E1 4.4063,E2 201.9431} C_DIS
LIN {X -57.1554,Y -121.7068,Z 182,A -111.0417,B 4.4552,C 0.3481,E1 4.402,E2 203.6212} C_DIS
LIN {X -59.8114,Y -120.4217,Z 182,A -112.4017,B 4.4552,C 0.3476,E1 4.3986,E2 204.9942} C_DIS
LIN {X -63.9166,Y -118.2961,Z 182,A -114.3713,B 4.4554,C 0.3452,E1 4.3937,E2 206.964} C_DIS
LIN {X -67.7507,Y -116.143,Z 182,A -116.3571,B 4.4555,C 0.3437,E1 4.3889,E2 208.964} C_DIS
LIN {X -71.4233,Y -113.9213,Z 182,A -118.1826,B 4.4557,C 0.3412,E1 4.3845,E2 210.7891} C_DIS
LIN {X -74.6179,Y -111.8542,Z 182,A -119.8141,B 4.4559,C 0.3389,E1 4.3807,E2 212.4219} C_DIS
LIN {X -78.2935,Y -109.313,Z 182,A -121.7349,B 4.4561,C 0.3361,E1 4.3763,E2 214.3447} C_DIS
LIN {X -81.8058,Y -106.71,Z 182,A -123.6354,B 4.4563,C 0.3334,E1 4.3721,E2 216.2498} C_DIS
LIN {X -85.0686,Y -104.1275,Z 182,A -125.4717,B 4.4565,C 0.3309,E1 4.3681,E2 218.0939} C_DIS
LIN {X -88.454,Y -101.2674,Z 182,A -127.3909,B 4.4567,C 0.3278,E1 4.364,E2 220.0167} C_DIS
LIN {X -91.8932,Y -98.1578,Z 182,A -129.3543,B 4.457,C 0.3241,E1 4.3599,E2 221.9783} C_DIS
LIN {X -94.5896,Y -95.5619,Z 182,A -131.0697,B 4.4571,C 0.322,E1 4.3565,E2 223.7085} C_DIS
LIN {X -97.5641,Y -92.5233,Z 182,A -132.887,B 4.4574,C 0.3185,E1 4.353,E2 225.5262} C_DIS
LIN {X -100.7391,Y -89.0552,Z 182,A -134.9517,B 4.4576,C 0.3149,E1 4.3491,E2 227.598} C_DIS
LIN {X -103.7643,Y -85.5118,Z 182,A -136.9905,B 4.4579,C 0.3111,E1 4.3454,E2 229.643} C_DIS
LIN {X -106.5275,Y -82.0442,Z 182,A -138.9612,B 4.4582,C 0.3076,E1 4.342,E2 231.6233} C_DIS
LIN {X -109.1983,Y -78.4539,Z 182,A -140.9091,B 4.4584,C 0.3036,E1 4.3388,E2 233.5758} C_DIS
LIN {X -111.2054,Y -75.5819,Z 182,A -142.3102,B 4.4587,C 0.2995,E1 4.3366,E2 234.9649} C_DIS
Enddeposition()
END
